nut_long  := 0.0;
nut_obliq := 0.0;

FOR i:=0 TO 62 DO
	nut_long  := nut_long  + 0.0001*( (sdelt[i]*t + sin_lng[i])*sarg[i]);
	nut_obliq := nut_obliq + 0.0001*( (cdelt[i]*t + cos_lng[i])*carg[i]);
END_FOR

END_FUNCTION_BLOCK

// ---- POUs/Functions/POLY.TcPOU
FUNCTION POLY : LREAL
VAR_INPUT
	// independent variable
	X:	LREAL;
END_VAR
VAR_IN_OUT
	// array of coefficients
	COEFFS: ARRAY [*] OF LREAL;
END_VAR
VAR
	i: DINT;
END_VAR

POLY := 0.0;
FOR i := LOWER_BOUND(COEFFS,1) TO UPPER_BOUND(COEFFS,1) DO
	POLY := POLY + COEFFS[i]*EXPT(X, i);
END_FOR

END_FUNCTION

// ---- POUs/FunctionBlocks/CO_ABERRATION.TcPOU
FUNCTION_BLOCK CO_ABERRATION
VAR_INPUT
	jd, 				// Julian Date
	ra, dec: LREAL; 	//ra and dec in degrees
	eps : LREAL := 0.0;
END_VAR
VAR_OUTPUT
	d_ra, d_dec: LREAL;
END_VAR
VAR
	sunpos: FB_SUNPOS;
	nutate: FB_NUTATE;
	sunra, sundec, sunlon,
	d_psi, d_epsilon, eps0,
	t, e, peri, cd, sd, ce, te, cp, sp, cs, ss, ca, sa, term1, term2, term3, term4: LREAL;
END_VAR
VAR CONSTANT
	d2r : LREAL := PI/180.0;
	k: LREAL := 20.49552; //constant of aberration, in arcseconds
	
END_VAR

(*
;+
;  NAME:
;     CO_ABERRATION
; PURPOSE:
;     Calculate changes to Ra and Dec due to the effect of annual aberration 
; EXPLANATION:
;      as described in Meeus, Chap 23.
; CALLING SEQUENCE:
;      co_aberration, jd, ra, dec, d_ra, d_dec, [EPS = ]
; INPUTS
;       jd      : Julian Date [scalar or vector]
;       ra, dec : Arrays (or scalars) of the ra  and dec's in degrees
;   Note: if jd is a vector, then ra and dec must either be scalars, or 
;                vectors of the same length.
;
; OUTPUTS
;       d_ra, d_dec: the corrections to ra and dec due to aberration in 
;                    arcseconds.  (These values can be added to the true RA 
;                    and dec to get the apparent position).   Note that d_ra
;                     is *not* multiplied by cos(dec), so that 
;                     apparent_ra = ra + d_ra/3600. 
; OPTIONAL INPUT KEYWORD:
;       eps : set this to the true obliquity of the ecliptic (in radians), or
;         it will be set for you if you don't know it (in that case, set it to
;                 an empty variable).
; EXAMPLE:
;   Compute the change in RA and Dec of Theta Persei (RA = 2h46m,11.331s, Dec =
;   49d20',54.54") due to aberration on 2028 Nov 13.19 TD
;
;      IDL> jdcnv,2028,11,13,.19*24,jd      ;Get Julian date
;      IDL> co_aberration,jd,ten(2,46,11.331)*15,ten(49,20,54.54),d_ra,d_dec
;
;      ==> d_ra = 30.045" (=2.003s)    d_dec = 6.697"
; NOTES:
;  These formula are from Meeus, Chapters 23.  Accuracy is much better than 1 
;   arcsecond.
;
;   The maximum deviation due to annual aberration is 20.49" and occurs when the
;   Earth velocity is perpendicular to the direction of the star.
;
; REVISION HISTORY:
;   Written, June 2002,      Chris O'Dell, U. of Wisconsin
;   Fix error with vector input   W. Landsman   June 2009
;   June 2009 update fixed case where JD was scalar but RA,Dec were vectors, but 
;     broke the case when both JD and RA,Dec were vectors Aug 2012 W. Landsman
;   Further fix when JD is 1 element vector  W. Landsman
;-
*)

T := (jd -2451545.0)/36525.0; // julian centuries from J2000 of jd.

IF EPS = 0.0 THEN
	// must calculate obliquity of ecliptic
	nutate(jd := jd, nut_long => d_psi, nut_obliq => d_epsilon); //d_psi and d_epsilon in degrees
	eps0 := ten(23,26,21.448)*3600.0 - 46.8150*T - 0.00059*EXPT(T, 2) +  0.001813*EXPT(T, 3);
	// TRUE obliquity OF the ecliptic in radians
	eps := (eps0 + d_epsilon)/3600.0*d2r; 	
END_IF

sunpos( JD := jd, RA => sunra, Dec => sundec, longmed => sunlon);

// Earth's orbital eccentricity
e := 0.016708634 - 0.000042037*T - 0.0000001267*EXPT(T, 2);
// longitude of perihelion, in degrees 
peri := 102.93735 + 1.71946*T + 0.00046*EXPT(T, 2);

//Useful Trig Functions
cd := COS(dec*d2r);		sd := SIN(dec*d2r);
ce := COS(eps); 		te := TAN(eps);
cp := COS(peri*d2r);	sp := SIN(peri*d2r);
cs := COS(sunlon*d2r);	ss := SIN(sunlon*d2r);
ca := COS(ra*d2r);		sa := SIN(ra*d2r);

term1 := (ca*cs*ce + sa*ss)/cd;
term2 := (ca*cp*ce + sa*sp)/cd;
term3 := (cs*ce*(te*cd - sa*sd) + ca*sd*ss);
term4 := (cp*ce*(te*cd - sa*sd) + ca*sd*sp);

d_ra := -k * term1 + e*k * term2;
d_dec := -k * term3 + e*k * term4;

END_FUNCTION_BLOCK

// ---- POUs/FunctionBlocks/FB_SUNPOS.TcPOU
FUNCTION_BLOCK FB_SUNPOS
VAR_INPUT
	// Julian Date
	JD:		LREAL;
	// output in Radians instead of Degrees
	RADIAN:	BOOL:= FALSE;
END_VAR
VAR_OUTPUT
	// right ascension
	RA,
	// declination of the sun
	Dec,
	// longitude
	longmed,
	// True Obliquity
	oblt:	LREAL;
END_VAR
VAR
	t, //  Julian centuries FROM 1900.0
	l, //  sun's mean longitude
	me, // Earth's mean anomaly
	ellcor, // ellipticity of the orbit
	mv, // mean anomaly of Venus
	vencorr,
	mm, 
	marscorr,
mj, jupcorr,
d, longterm, mooncorr,  omega:	LREAL;
END_VAR
VAR CONSTANT
	dtor: LREAL := PI/180.0; // Pi/180
END_VAR

(* source: https://idlastro.gsfc.nasa.gov/ftp/pro/astro/sunpos.pro *)

//  form TIME in Julian centuries FROM 1900.0
t := (jd - 2415020.0)/36525.0;

//  form sun's mean longitude
l := (279.696678+LMOD(36000.768925*t, 360.0))*3600.0;

//  allow for ellipticity of the orbit (equation of centre) using the Earth's mean anomaly ME
me := 358.475844 + LMOD(35999.049750*t, 360.0);
ellcor  := (6910.1 - 17.2*t)*SIN(me*dtor) + 72.3*SIN(2.0*me*dtor);
l := l + ellcor;
 
// allow FOR the Venus perturbations using the mean anomaly OF Venus MV
mv := 212.603219 + LMOD(58517.803875*t, 360.0);
vencorr := 4.8 * COS((299.1017 + mv - me)*dtor) + 
          5.5 * COS((148.3133 +  2.0 * mv  -  2.0 * me )*dtor) + 
          2.5 * COS((315.9433 +  2.0 * mv  -  3.0 * me )*dtor) + 
          1.6 * COS((345.2533 +  3.0 * mv  -  4.0 * me )*dtor) + 
          1.0 * COS((318.15   +  3.0 * mv  -  5.0 * me )*dtor);
l := l + vencorr;

//  Allow FOR the Mars perturbations using the mean anomaly OF Mars MM
mm := 319.529425  +  LMOD( 19139.858500 * t,  360.0 );
marscorr := 2.0 * COS((343.8883 -  2.0 * mm  +  2.0 * me)*dtor ) + 
            1.8 * COS((200.4017 -  2.0 * mm  + me) * dtor);
l := l + marscorr;

// Allow FOR the Jupiter perturbations using the mean anomaly OF Jupiter MJ
mj := 225.328328  +  LMOD( 3034.6920239 * t,  360.0 );
jupcorr := 7.2 * COS(( 179.5317 - mj + me )*dtor) + 
          2.6 * COS((263.2167  -  MJ ) *dtor) + 
          2.7 * COS(( 87.1450  -  2.0 * mj  +  2.0 * me ) *dtor) + 
          1.6 * COS((109.4933  -  2.0 * mj  +  me ) *dtor);
l := l + jupcorr;

// Allow FOR the Moons perturbations using the mean elongation OF the Moon from the Sun D
d := 350.7376814  + LMOD( 445267.11422 * t,  360.0 );
mooncorr  := 6.5 * SIN(d*dtor);
l := l + mooncorr;

// Allow for long period terms
longterm := 6.4 * SIN(( 231.19  +  20.20 * t )*dtor);
l :=  l + longterm;
l :=  LMOD( l + 2592000.0,  1296000.0); 
longmed := l/3600.0;

// Allow for Aberration
l :=  l - 20.5;

// Allow for Nutation using the longitude of the Moons mean node OMEGA
omega := 259.183275 - LMOD( 1934.142008 * t, 360.0);
l :=  l - 17.2 * SIN(omega*dtor);

// Form the True Obliquity
oblt := 23.452294 - 0.0130125*t + (9.2*COS(omega*dtor))/3600.0;

// Form Right Ascension AND Declination
l := l/3600.0;
//ra := ATAN2( COS(l*dtor), SIN(l*dtor) * COS(oblt*dtor));
ra := ATAN2( SIN(l*dtor) * COS(oblt*dtor), COS(l*dtor));
dec := ASIN(SIN(l*dtor) * SIN(oblt*dtor));
 
IF RADIAN THEN
	oblt := oblt*dtor; 
	longmed := longmed*dtor;
ELSE // result in degrees
	ra := MODABS(ra/dtor, 360.0);
    dec := dec/dtor;
END_IF

END_FUNCTION_BLOCK

// ---- POUs/Functions/TEN.TcPOU
FUNCTION TEN : LREAL
VAR_INPUT
	dd,mm,ss: LREAL;
END_VAR
VAR
END_VAR

TEN := dd + (mm/60.0) + (ss/3600.0);

END_FUNCTION

// ---- POUs/FunctionBlocks/CO_REFRACT.TcPOU
FUNCTION_BLOCK CO_REFRACT
VAR_INPUT
	old_alt: LREAL;
	altitude: LREAL := 0.0;
	pressure: LREAL := 0.0;
	temperature: LREAL := 0.0;
	epsilon: LREAL := 0.25; //accuracy of iteration for observed=TRUE case, in arcseconds
	TO_OBSERVED: BOOL;
END_VAR
VAR_OUTPUT
	new_alt: LREAL;
END_VAR
VAR
	aout, P, T, dr, cur, last : LREAL;
END_VAR
VAR CONSTANT
	alpha : LREAL := 0.0065; //temp lapse rate [deg C per meter]
END_VAR

IF temperature = 0.0 THEN
	IF altitude > 11000.0 THEN 
		temperature := 211.5; 
	ELSE 
		temperature := 283.0 - alpha*altitude;
	END_IF
END_IF

// estimate Pressure based on altitude, using U.S. Standard Atmosphere formula.
IF pressure = 0 THEN 
	pressure := 1010.0*EXPT(1-6.5/288000*altitude, 5.255);
END_IF

IF NOT TO_OBSERVED THEN 
	aout := old_alt - co_refract_forward(old_alt, P:=pressure,T:=temperature);
ELSE
	aout := 0.0;
	P := pressure; T := temperature;
	//calculate initial refraction guess
	dr := co_refract_forward(old_alt, P:=P, T:=T);
	cur := old_alt + dr; // guess of observed location

	REPEAT 
	 	last := cur;
		dr := co_refract_forward(cur, P:= P, T:=T);
	  	cur := old_alt + dr;
	UNTIL ABS(last-cur)*3600.0 < epsilon
	END_REPEAT
	aout := cur;
END_IF

new_alt := aout;

END_FUNCTION_BLOCK

// ---- POUs/Functions/CO_REFRACT_FORWARD.TcPOU
FUNCTION CO_REFRACT_FORWARD : LREAL
VAR_INPUT
	// The observed (apparent) altitude, in DEGREES.
	a: LREAL;
	// Pressure [in millibars]. Default is 1010 millibars.
	P: LREAL := 1010.0;
	// Ground Temp [in Celsius].  Default is 0 Celsius.
	T: LREAL := 0.0;
END_VAR
VAR
	Ref, tpcor: LREAL;
END_VAR
VAR CONSTANT
	d2r : LREAL := PI/180.0;
END_VAR

a := LIMIT(0.0, a, 90.0);
P := LIMIT(600.0, P, 1200.0);
T := LIMIT(-40.0, T, 40.0);

IF a >= 15.0 THEN
	Ref := 1.0 / TAN((a + 7.31/(a+4.4))*d2r);
ELSE
	Ref := 3.569*(0.1594 + 0.0196*a + 0.00002*EXPT(a, 2))/(1.0+0.505*a + 0.0845*EXPT(a, 2));
END_IF
tpcor := P * 283.15 / (1010.0 * (273.15 + T));
CO_REFRACT_FORWARD := tpcor * Ref;

END_FUNCTION

// ---- POUs/FunctionBlocks/FB_PRECESS.TcPOU
FUNCTION_BLOCK FB_PRECESS
VAR_INPUT
	ra, 
	dec,
	equinox1,
	equinox2: LREAL;
	RADIAN:	BOOL := FALSE;
END_VAR
VAR_OUTPUT
	ra_precessed,
	dec_precessed:	LREAL;
END_VAR
VAR
	ra_rad, dec_rad: LREAL;
	a,b,c,t: LREAL;
	x, x2: ARRAY[0..2] OF LREAL;
	st1: LREAL;
	rot: ARRAY[0..2,0..2] OF LREAL;
	sina, sinb, sinc, cosa,cosb,cosc: LREAL;
END_VAR
VAR CONSTANT
	deg_to_rad : LREAL := PI/180.0;
	sec_to_rad : LREAL := deg_to_rad/3600.0;
END_VAR

IF NOT RADIAN THEN
	ra_rad := ra*deg_to_rad;
	dec_rad := dec*deg_to_rad;
ELSE
    //Convert TO double precision IF NOT already
	ra_rad := ra;
	dec_rad := dec;
END_IF

a := COS( dec_rad );
x[0] := a*COS(ra_rad); x[1] := a*SIN(ra_rad); x[2] := SIN(dec_rad);

//*** PREMAT code starts here
ST1 := 0.001*( equinox1 - 2000.0);
t := 0.001*( equinox2 - equinox1);
//  Compute 3 rotation angles
A := sec_to_rad * T * (23062.181 + ST1*(139.656 +0.0139*ST1) + T*(30.188 - 0.344*ST1+17.998*T));
B := sec_to_rad * T * T * (79.280 + 0.410*ST1 + 0.205*T) + A;
C := sec_to_rad * T * (20043.109 - ST1*(85.33 + 0.217*ST1) + T*(-42.665 - 0.217*ST1 -41.833*T));
  sina := SIN(a); sinb := SIN(b);  sinc := SIN(c);
  cosa := COS(a); cosb := COS(b);  cosc := COS(c);

rot[0,0] :=  cosa*cosb*cosc-sina*sinb; 	rot[0,1] := sina*cosb+cosa*sinb*cosc; 	rot[0,2] := cosa*sinc;
rot[1,0] := -cosa*sinb-sina*cosb*cosc; 	rot[1,1] := cosa*cosb-sina*sinb*cosc; 	rot[1,2] := -sina*sinc;
rot[2,0] := -cosb*sinc;					rot[2,1] := -sinb*sinc; 				rot[2,2] := cosc;

//*** PREMAT code ends here

//x2 := rot* x; //rotate to get output direction cosines
x2[0] := rot[0,0]*x[0] + rot[1,0]*x[1] + rot[2,0]*x[2];
x2[1] := rot[0,1]*x[0] + rot[1,1]*x[1] + rot[2,1]*x[2];
x2[2] := rot[0,2]*x[0] + rot[1,2]*x[1] + rot[2,2]*x[2];

ra_rad := atan2(x2[1],x2[0]);
dec_rad := ASIN(x2[2]);

IF NOT RADIAN THEN
	ra_precessed := ra_rad/deg_to_rad;
	ra_precessed := MODABS(ra_precessed, 360.0);            //RA between 0 AND 360 degrees
	dec_precessed := dec_rad/deg_to_rad;
ELSE
	ra_precessed := ra_rad; 
	dec_precessed := dec_rad;
	ra_precessed := MODABS(ra_rad, 2.0*PI);
END_IF

END_FUNCTION_BLOCK

// ---- POUs/FunctionBlocks/FB_ALTAZ2HADEC.TcPOU
FUNCTION_BLOCK FB_ALTAZ2HADEC
VAR_INPUT
	// the local apparent altitude, in DEGREES
	alt:	LREAL;
	// the local apparent azimuth, in DEGREES
	az:		LREAL;
	// the local geodetic latitude, in DEGREES
	lat: 	LREAL;
END_VAR
VAR_OUTPUT
	// the local apparent hour angle, in DEGREES
	ha:		LREAL;
	// the local apparent declination, in DEGREES
	dec:	LREAL;
END_VAR
VAR
	alt_r:	LREAL;
	az_r:	LREAL;
	lat_r:	LREAL;
	sindec: LREAL;
END_VAR
VAR CONSTANT
	d2r:	LREAL := PI/180.0;
	//r2d:	LREAL := 180.0/PI;
	//h2r:	LREAL := PI/12.0;
	//h2d:	LREAL := 15.0;
END_VAR

(*

  NAME:
    ALTAZ2HADEC
 PURPOSE:
    Convert Horizon (Alt-Az) coordinates to Hour Angle and Declination.
 EXPLANATION::
    Can deal with the NCP singularity.    Intended mainly to be used by
    program hor2eq.pro
 CALLING SEQUENCE:
   ALTAZ2HADEC, alt, az, lat, ha, dec

 INPUTS
   alt - the local apparent altitude, in DEGREES, scalar or vector
   az  - the local apparent azimuth, in DEGREES, scalar or vector,
         measured EAST of NORTH!!!  If you have measured azimuth west-of-south
        (like the book MEEUS does), convert it to east of north via:
                       az = (az + 180) mod 360

   lat -  the local geodetic latitude, in DEGREES, scalar or vector.

 OUTPUTS
   ha  -  the local apparent hour angle, in DEGREES.  The hour angle is the 
          time that right ascension of 0 hours crosses the local meridian.  
          It is unambiguously defined.
   dec -  the local apparent declination, in DEGREES.

 EXAMPLE:
     Arcturus is observed at an apparent altitude of 59d,05m,10s and an 
     azimuth (measured east of north) of 133d,18m,29s while at the 
     latitude of +43.07833 degrees.
     What are the local hour angle and declination of this object?

     IDL> altaz2hadec, ten(59,05,10), ten(133,18,29), 43.07833, ha, dec
     ===> Hour angle ha = 336.683 degrees
          Declination, dec = 19.1824 degrees

       The widely available XEPHEM code gets:
                 Hour Angle = 336.683
                 Declination = 19.1824

 REVISION HISTORY:
    Written  Chris O'Dell Univ. of Wisconsin-Madison May 2002
*)
alt_r  := alt*d2r;
az_r := az*d2r;
lat_r := lat*d2r;

//******************************************************************************
// find local HOUR ANGLE (in degrees, from 0. to 360.)
ha := atan2( -SIN(az_r)*COS(alt_r), 
           -COS(az_r)*SIN(lat_r)*COS(alt_r)+SIN(alt_r)*COS(lat_r));
ha := ha / d2r;
IF ha < 0.0 THEN 
	ha := ha + 360.0;
END_IF
 ha := MODABS(ha, 360.0);

// Find declination (positive if north of Celestial Equator, negative if south)
sindec := SIN(lat_r)*SIN(alt_r) + COS(lat_r)*COS(alt_r)*COS(az_r);
// convert dec to degrees
dec := ASIN(sindec)/d2r;

END_FUNCTION_BLOCK

// ---- POUs/Functions/CT2LST.TcPOU
FUNCTION CT2LST : LREAL
VAR_INPUT
	lng: LREAL; // The longitude in degrees (east of Greenwich) of the place for which the local sidereal time is desired, scalar.   The Greenwich mean sidereal time (GMST) can be found by setting Lng = 0.
	jd:	LREAL; // this is the Julian date of time in question
END_VAR
VAR
	t0,t,theta: LREAL;
END_VAR
VAR CONSTANT
	jd2000: LREAL := 2451545.0;
END_VAR

(* source https://idlastro.gsfc.nasa.gov/ftp/pro/astro/ct2lst.pro 

;+
; NAME:
;     CT2LST
; PURPOSE:
;     To convert from Local Civil Time to Local Mean Sidereal Time.
;
; CALLING SEQUENCE:
;     CT2LST, Lst, Lng, Tz, Time, [Day, Mon, Year] 
;                       or
;     CT2LST, Lst, Lng, dummy, JD
;
; INPUTS:
;     Lng  - The longitude in degrees (east of Greenwich) of the place for 
;            which the local sidereal time is desired, scalar.   The Greenwich 
;            mean sidereal time (GMST) can be found by setting Lng = 0.
;     Tz  - The time zone of the site in hours, positive East  of the Greenwich
;           meridian (ahead of GMT).  Use this parameter to easily account 
;           for Daylight Savings time (e.g. -4=EDT, -5 = EST/CDT), scalar
;           This parameter is not needed (and ignored) if Julian date is 
;           supplied.    ***Note that the sign of TZ was changed in July 2008
;           to match the standard definition.*** 
;     Time or JD  - If more than four parameters are specified, then this is 
;               the time of day of the specified date in decimal hours.  If 
;               exactly four parameters are specified, then this is the 
;               Julian date of time in question, scalar or vector
;
; OPTIONAL INPUTS:
;      Day -  The day of the month (1-31),integer scalar or vector
;      Mon -  The month, in numerical format (1-12), integer scalar or vector
;      Year - The 4 digit year (e.g. 2008), integer scalar or vector
;
; OUTPUTS:
;       Lst   The Local Sidereal Time for the date/time specified in hours.
;
; RESTRICTIONS:
;       If specified, the date should be in numerical form.  The year should
;       appear as yyyy.
;
; PROCEDURE:
;       The Julian date of the day and time is question is used to determine
;       the number of days to have passed since 0 Jan 2000.  This is used
;       in conjunction with the GST of that date to extrapolate to the current
;       GST; this is then used to get the LST.    See Astronomical Algorithms
;       by Jean Meeus, p. 84 (Eq. 11-4) for the constants used.
;
; EXAMPLE:
;       Find the Greenwich mean sidereal time (GMST) on 2008 Jul 30 at 15:53 pm
;       in Baltimore, Maryland (longitude=-76.72 degrees).   The timezone is 
;       EDT or tz=-4
;
;       IDL> CT2LST, lst, -76.72, -4,ten(15,53), 30, 07, 2008
;
;               ==> lst =  11.356505  hours  (= 11h 21m 23.418s)
;
;       The Web site  http://tycho.usno.navy.mil/sidereal.html contains more
;       info on sidereal time, as well as an interactive calculator.
; PROCEDURES USED:
;       jdcnv - Convert from year, month, day, hour to julian date
;
; MODIFICATION HISTORY:
;     Adapted from the FORTRAN program GETSD by Michael R. Greason, STX, 
;               27 October 1988.
;     Use IAU 1984 constants Wayne Landsman, HSTX, April 1995, results 
;               differ by about 0.1 seconds  
;     Longitudes measured *east* of Greenwich   W. Landsman    December 1998
;     Time zone now measure positive East of Greenwich W. Landsman July 2008
;     Remove debugging print statement  W. Landsman April 2009
;-

*)

t0 := jd - jd2000;
t := t0/36525.0;
// Compute GST in seconds.
theta := 280.46061837 + (360.98564736629 * t0) + EXPT(t, 2)*(0.000387933 - (t/ 3871.0E4));
//theta := 100.46061837 + 36000.770053608*t0 + 0.000387933*EXPT(t0,2) - EXPT(t0,3)/3871000.0;
// Compute LST in hours.
CT2LST := ( theta + lng)/15.0;
CT2LST := MODABS(CT2LST, 24.0);

END_FUNCTION

// ---- POUs/TelescopeAuxiliary.TcPOU
PROGRAM TelescopeAuxiliary
VAR
	MQTTTimer : TON := (PT:=T#5S);
	pressure_voltage:	REAL;
END_VAR
VAR_OUTPUT
	// BT9 mirror
	temperature_mirror2:	REAL;
	// BT10
	temperature_mirror1:	REAL;
	// BT11

	// dewar pressure 0..10V Pfeiffer 
	pressure_Dewar:	REAL;
	// dewar temperature PT100
	temperature_Dewar:	REAL;
	

END_VAR

temperature_mirror2 := GVL_Telescope.temperature_mirror2 / 100.0;
temperature_mirror1 := GVL_Telescope.temperature_mirror1 / 100.0;

MQTTTimer(IN:=TRUE);
IF MQTTTimer.Q THEN // publish new payload every second

	MAIN.MQTTClient.Publish('telescope', 'dome',  'Mirror2Temperature',	LREAL_TO_FMTSTR(temperature_mirror2, 2, TRUE));
	MAIN.MQTTClient.Publish('telescope', 'dome', 'Mirror1Temperature',	LREAL_TO_FMTSTR(temperature_mirror1, 2, TRUE));
	
	MAIN.MQTTClient.Publish('telescope', 'instrument', 'DewarPressureVoltage',	LREAL_TO_FMTSTR(pressure_voltage, 3, TRUE));
	IF NOT GVL_Auxiliary.Dewar_temperature_error THEN
		MAIN.MQTTClient.Publish('telescope', 'instrument', 'DewarTemperature',	LREAL_TO_FMTSTR(temperature_Dewar, 2, TRUE));
	END_IF
	IF pressure_voltage > 0.001 THEN
		MAIN.MQTTClient.Publish('telescope', 'instrument', 'DewarPressure',	LREAL_TO_FMTSTR(pressure_Dewar, 2, TRUE));
	END_IF
	
	MQTTTimer(IN:=FALSE);

END_IF

END_PROGRAM

// ---- POUs/Functions/DateTime2JD.TcPOU
FUNCTION DateTime2JD : LREAL
VAR_INPUT
	epoch: TIMESTRUCT;
END_VAR
VAR
	a,y,m,d,jdn: LREAL;
END_VAR

(*    import datetime
    from math import floor
    if not type(epoch) is datetime.datetime:
        raise TypeError('datetime must be of type datetime')
    
    a = floor((14 - epoch.month)/12)
    y = epoch.year + 4800 - a
    m = epoch.month + 12*a - 3
    
    d = epoch.day
    d += epoch.hour/24. + epoch.minute/1440. + epoch.second/86400. # microsecond might be added here?
    
    if [epoch.year,epoch.month,d] >= [1582,10,15]:
        jdn = epoch.day + floor((153*m + 2)/5) + 365*y + floor(y/4) - floor(y/100) + floor(y/400) - 32045
    elif [epoch.year,epoch.month,d] <= [1582,10,4]:
        jdn = epoch.day + floor((153*m + 2)/5) + 365*y + floor(y/4) - 32083
    return jdn + (epoch.hour-12)/24. + epoch.minute/1440. + epoch.second/86400.
*)
a := FLOOR((14.0 - epoch.wMonth)/12.0);
y := epoch.wYear + 4800.0 - a;
m := epoch.wMonth + 12.0*a - 3.0;

d := epoch.wDay + (epoch.wHour/24.0) + (epoch.wMinute/1440.0) + (epoch.wSecond/86400.0);

//IF (epoch.wYear > 1582) (* AND (epoch.wMonth > 10.0) AND (d > 15.0)*) THEN
	jdn := epoch.wDay + FLOOR((153*m + 2)/5) + 365.0*y + FLOOR(y/4) - FLOOR(y/100) + FLOOR(y/400) - 32045.0;
//ELSIF (epoch.wYear < 1582) AND (epoch.wMonth < 10) AND (d > 4.0) THEN
//	jdn := epoch.wDay + FLOOR((153*m + 2)/5) + 365.0*y + FLOOR(y/4) - 32083.0;
//END_IF

DateTime2JD := jdn
			+ (epoch.wHour-12.0)/24.0
			+ (epoch.wMinute/1440.0) 
			+ (epoch.wSecond/86400.0)
			+ (DWORD_TO_REAL(epoch.wMilliseconds)/86400000.0);

END_FUNCTION

// ---- POUs/ElevationControl.TcPOU
PROGRAM ElevationControl
VAR_INPUT
	// increase the eleveation
	up:			BOOL;
	// decrease the elevation
	down:		BOOL;
	// reset an error
	reset:		BOOL;
	// enable the axis
	enable: 	BOOL;
	// set position of the axis in degrees
	position:	LREAL;
	// move axis command
	MoveAxis:	BOOL;
	// calibrate the focus axis
	HomeAxis:	BOOL;
	// enable tracking
	Tracking:	BOOL;
END_VAR
VAR_OUTPUT
	// axis is ready to operate
	Ready:			BOOL;
	// drive error condition
	error: 			BOOL;
	// warning condition
	warning:		BOOL;
	// actual position of the elevation axis
	act_position: 	LREAL;
	// error ID of the elevation axis
	ErrorID: 		UDINT;
	// axis is calibrated
	Calibrated:		BOOL;
	// time to reach target position
	slewtime:		LREAL;
END_VAR
VAR
	ElevationAxis:			FB_Axis2;
	ElevationCalibration: 	MC_SetPosition;
	fbSoEReset: 			FB_SoEReset;
	bSoEReset : BOOL;
	// delay until commutator angle is measured
	readydelay:				TON;
	getlastposition:		BOOL := TRUE;
	ElevationAxisEvent: 	FB_Eventlog;
	ElevationBrakeEvent: 	FB_Eventlog;
	HighElevationEvent: 	FB_Eventlog;
	LowElevationEvent:		FB_Eventlog;
	TorqueWarning:			FB_EventLog;
	CalibrationEvent:		FB_Eventlog;
	elevation_torque: REAL;
	ReadParameter:		MC_ReadParameter;
END_VAR
VAR CONSTANT
	// current position of the calibration cam. Apply an offset here if necessary
	calibration_position:	LREAL := 45.0;
END_VAR
VAR PERSISTENT
	last_position:	LREAL := -1.0;
END_VAR

// limit the position input to a sane value
position := LIMIT(0.0, position, 90.0);

//if we enable the axis, we have to open the brake first
IF Enable THEN
	HydraulicsControl.open_brake := TRUE;
END_IF

// if an error occurs on te enabled axis we close the brake
IF Enable AND error THEN
	Enable := FALSE;
	HydraulicsControl.close_brake := TRUE;
END_IF

IF ElevationAxis.Calibrated OR Error THEN
	HomeAxis := FALSE;
END_IF

Calibrated := ElevationAxis.Calibrated;

IF HomeAxis THEN
//	position := homing_position;
	position := calibration_position;
	MoveAxis := FALSE;
	Tracking := FALSE;
END_IF

IF MoveAxis THEN
	Tracking := FALSE;
END_IF

// if NOT Enabled and ActVelo>1 then issue a warning
warning := NOT enable AND GVL_Telescope.ElevationAxisRef.NcToPlc.ActVelo>2.0;

// deactivate limit switches on homing
MC_SetAcceptBlockedDriveSignal(
	Axis := GVL_Telescope.ElevationAxisRef, 
	Enable := HomeAxis);

IF Tracking AND ABS(position - act_position) > 1.0 THEN
	MoveAxis := TRUE;
END_IF

	
ElevationAxis(
	Enable := 			enable AND HydraulicsControl.brake_open,
	Reset := 			reset,
	MoveAxis :=			MoveAxis,
	HomeAxis :=			HomeAxis,
	Tracking :=			Tracking,
	Position := 		position, 
	Enable_Positive :=  GVL_Telescope.Elevation_inputs.0 OR HomeAxis,
	Enable_Negative := 	GVL_Telescope.Elevation_inputs.1,
	Jog_Forward :=		up,
	Jog_Backwards := 	down,
	bCalibrationCam :=	NOT GVL_Telescope.Elevation_inputs.0,
	ActualPosition => 	act_position,
	Error => 			error,
	ErrorID => 			ErrorID,
	AxisRef :=			GVL_Telescope.ElevationAxisRef);

IF ElevationAxis.MoveDone THEN
	MoveAxis := FALSE;
END_IF

IF ElevationAxis.HomeDone THEN
	HomeAxis := FALSE;
END_IF
	
IF ElevationAxis.ResetDone THEN
	reset := FALSE;
END_IF

ElevationCalibration(Axis := GVL_Telescope.ElevationAxisRef,
	Execute := getlastposition AND last_position>=0.0 AND NOT Calibrated,
	Position := last_position);

IF ElevationCalibration.Done THEN
	getlastposition := FALSE;
END_IF

IF Calibrated THEN
	last_position := act_position;
END_IF
	
bSoEReset := GVL_Telescope.Elevation_diagnostic = 16#0000F10B OR GVL_Telescope.Elevation_diagnostic = 16#0000F601;

IF bSoEReset THEN
	last_position := -1.0;
	fbSoEReset(
		Axis := GVL_Telescope.ElevationAxisRef,
		Execute := TRUE,
		Timeout := DEFAULT_ADS_TIMEOUT);
 	IF NOT fbSoEReset.Busy THEN
		fbSoEReset(Axis := GVL_Telescope.ElevationAxisRef, Execute := FALSE);
		bSoEReset := FALSE;
		Reset := TRUE;
	END_IF
END_IF 

readydelay(IN :=  HydraulicsControl.brake_open, PT := T#6000MS, Q=> ready);

ReadParameter(	Axis := GVL_Telescope.ElevationAxisRef, 
				Enable := ElevationAxis.InMotion, 
				ParameterNumber := MC_AxisParameter.AxisRemainingTimeToGo, 
				ReadMode := E_ReadMode.READMODE_CYCLIC);
				
IF ReadParameter.Valid THEN
	slewtime := ReadParameter.Value;
END_IF

elevation_torque := GVL_Telescope.Elevation_torque / 10.0;

		
ElevationAxisEvent(	Trigger := Error, 
				Level := ADSLOG_MSGTYPE_ERROR,
				FormatString := 'Elevation Axis Error: %s',
				OnMessage := NCError_TO_STRING(ErrorID));

HighElevationEvent(	Trigger := Calibrated AND act_position > 80.0, 
				Level := ADSLOG_MSGTYPE_WARN,
				FormatString := 'High Elevation: %s',
				OnMessage := LREAL_TO_FMTSTR(act_position, 2, TRUE));

LowElevationEvent(	Trigger := Calibrated AND act_position < 15.0, 
				Level := ADSLOG_MSGTYPE_WARN,
				FormatString := 'Low Elevation: %s',
				OnMessage := LREAL_TO_FMTSTR(act_position, 2, TRUE));
				
ElevationBrakeEvent( Trigger := NOT enable AND HydraulicsControl.brake_open, 
				Level := ADSLOG_MSGTYPE_WARN,
				FormatString := '%s',
				OnMessage := 'Brake was opened without elevation axis enabled!'); 

TorqueWarning(	
	Trigger := 		ABS(elevation_torque) > 60.0, 
	Level := 		ADSLOG_MSGTYPE_WARN,
	FormatString :=	'%s',
	OnMessage := 	'Elevation torque is high.');
	
CalibrationEvent(
	Trigger :=	Calibrated,
	Level :=	ADSLOG_MSGTYPE_HINT,
	OnMessage := 'Elevation is calibrated.'
	);

END_PROGRAM

// ---- POUs/FunctionBlocks/FB_Axis2.TcPOU
FUNCTION_BLOCK FB_Axis2
VAR_INPUT
	// enable the axis
	Enable:		BOOL;
	// reset the axis after error
	Reset: 		BOOL;
	// Move the Axis to a given position
	MoveAxis: 	BOOL;
	// HomeAxis;
	HomeAxis:	BOOL;
	// Stop the axis
	StopAxis:	BOOL;
	// position to move to
	Position: 	LREAL;
	// maximum velocity
	Velocity:	LREAL := 10.0;
	// Enable movement in positive direction (considering limit switch)
	Enable_Positive:	BOOL := TRUE;
	// Enable movement in negative direction (considering limit switch)
	Enable_Negative:	BOOL := TRUE;
	// jog forward
	Jog_Forward:		BOOL := FALSE;
	// jog backward
	Jog_Backwards:		BOOL := FALSE;
	// calibration input for homing
	bCalibrationCam:	BOOL;
	isModuloAxis:		BOOL := FALSE;
	// enable external setpoint generator
	Tracking:			BOOL;
	HomingMode:			MC_HomingMode := MC_HomingMode.MC_DefaultHoming;
END_VAR
VAR_OUTPUT
	// Reset has been executed
	ResetDone:	BOOL; 
	// the axis is in target position
	MoveDone:	BOOL;
	// the axis hass jogged
	JogDone:	BOOL;
	// the axis has stopped
	StopDone: 	BOOL;
	// the axis was calibrated and has come to a standstill
	HomeDone:	BOOL;
	// the axis is ready
	Ready:		BOOL;
	// the command has been aborted
	CommandAborted: BOOL;
	// axis busy
	Busy: 		BOOL;
	// axis is moving
	Active: 	BOOL;
	// axis is stopping
	Stopping:	BOOL;
	// axis is standing still (no commands issued) this should be the default
	StandStill:	BOOL;
	// axis is in motion
	InMotion:	BOOL;
	// axis is homing
	Homing:		BOOL;
	// axis is Accelerating or Decelerating
	InRamp:		BOOL;
	// axis is tracking on position
	isTracking:	BOOL;
	//	error condition
	Error: 		BOOL;
	// number of error
	ErrorID: 	UDINT;
	// actual position of the axis
	ActualPosition: LREAL;
	// axis is calibrated;
	Calibrated:	BOOL := FALSE;
	
END_VAR
VAR
	Axis_Power:		MC_Power;
	Axis_Reset:		MC_Reset;
	Axis_Move:		MC_MoveAbsolute;
	Axis_Modulo:	MC_MoveModulo;
	//Axis_Position:	MC_ReadActualPosition;
	Axis_Stop:		MC_Stop;
	Axis_Status:	MC_ReadStatus;
	Axis_Home:		MC_Home;
	Axis_Jog: 		MC_Jog;
	Axis_SetpointEnable:	MC_ExtSetPointGenEnable;
	Axis_SetpointDisable:	MC_ExtSetPointGenDisable;
	StopAllowed:	BOOL;
	// Direction for Axis_SetpointFeed
	Direction:			DINT;
	// difference between set position and measured position
	PositionDifference:	LREAL;
	TrackPosition:		LREAL;
	TrackVelocity:		LREAL;
	TrackAcceleration:	LREAL;
END_VAR

VAR_IN_OUT
	// axis reference
	AxisRef:	AXIS_REF;
END_VAR

// query the status of the axis at the beginning of the cycle
Axis_Status(Enable := TRUE,
			Axis := AxisRef);

// Enable the axis (power signal or manual enable)
Axis_Power(
	Axis := AxisRef,
	Enable := Enable,
	Enable_Positive := Enable_Positive,
	Enable_Negative := Enable_Negative,
	Override := 100.0,
	Status => Ready);

Axis_Reset(
	Axis := 	AxisRef,
	Execute := 	Reset,
	Done => 	ResetDone);

(* Tracking section ********************************************** *)

IF Tracking THEN
	PositionDifference := LIMIT(-0.002, Position - ActualPosition, 0.002);
	TrackPosition := ActualPosition + PositionDifference;
	TrackVelocity := 0.0; // LIMIT(-1.0, 2.0 * Velocity, 1.0);
	TrackAcceleration := 0.0;
ELSE
	TrackPosition := ActualPosition;
	TrackVelocity := 0.0;
	TrackAcceleration := 0.0;
END_IF


IF NOT Tracking OR ABS(PositionDifference) < 1E-5 THEN // TrackVelocity = 0 AND TrackAcceleration = 0 THEN
	Direction := 0;
ELSIF PositionDifference < 0.0 THEN
	Direction := -1;
ELSE
	Direction := 1;
END_IF

isTracking := Tracking AND ABS(Position - ActualPosition) < 5.0E-3;
IF Tracking AND Ready AND Calibrated AND NOT StopAxis THEN
	Axis_SetpointEnable.Execute := TRUE;
ELSIF NOT Axis_SetpointEnable.Busy AND Axis_SetpointEnable.Done THEN
	Axis_SetpointEnable.Execute := FALSE;
END_IF

Axis_SetpointEnable(Axis := AxisRef,
	Position :=		TrackPosition,	// final destination
	PositionType := POSITIONTYPE_ABSOLUTE);
	
MC_ExtSetPointGenFeed(
	Position :=		TrackPosition,
	Velocity :=		TrackVelocity,
	Acceleration :=	TrackAcceleration,
	Direction :=	Direction, 
	Axis :=			AxisRef);

Axis_SetpointDisable(Axis := AxisRef,
	Execute := NOT Tracking);
	
(* end of tracking section  ********************************************** *)
	
IF isModuloAxis THEN
	Axis_Modulo( 
		Axis := 		AxisRef,
		Execute := 		MoveAxis AND Ready AND Calibrated,
		Position := 	Position,
		Velocity :=		Velocity,
		Direction := 	MC_Shortest_Way,
		Done => 		MoveDone);
ELSE
	Axis_Move( 
		Axis := 		AxisRef,
		Execute := 		MoveAxis AND Ready AND Calibrated,
		Position := 	Position,
		Velocity := 	Velocity,
		Done => 		MoveDone);
END_IF

Axis_Jog(
	JogForward := 	Jog_Forward AND Ready AND Enable_Positive,
	JogBackwards := Jog_Backwards AND Ready AND Enable_Negative,
	Mode := 		MC_JOGMODE_STANDARD_FAST,
	Done => 		JogDone, 
	Axis := 		AxisRef);

Axis_Home(
	Axis := 			AxisRef,
	Execute := 			HomeAxis AND Ready,
	Position := 		position, //DEFAULT_HOME_POSITION,
	HomingMode :=		HomingMode,
	bCalibrationCam := 	bCalibrationCam,
	Done => 			HomeDone);	
(*	
IF (MoveDone OR HomeDone OR JogDone) AND NOT Axis_Status.StandStill THEN
	StopAxis := TRUE;
END_IF
*)
IF MoveDone AND (NOT Axis_Modulo.Busy OR NOT Axis_Move.Busy) THEN
	MoveAxis := FALSE;
END_IF

IF JogDone THEN
	Jog_Forward := FALSE;
	Jog_Backwards := FALSE;
END_IF

IF HomeDone THEN
	Calibrated := TRUE;
	HomeAxis := FALSE;
END_IF

IF StopDone THEN
	StopAxis := FALSE;
END_IF

StopAllowed :=	Axis_Status.StandStill OR  
				Axis_Status.ContinuousMotion OR
				Axis_Status.DiscreteMotion OR
				Axis_Status.SynchronizedMotion OR
				Axis_Status.Homing;

Axis_Stop( 
	Axis := 	AxisRef,
	Execute := 	StopAxis AND StopAllowed,
	Done => 	StopDone);
(*
Axis_Position(
	Axis := 	AxisRef,
	Enable := 	Calibrated,
	Position => AbsolutePosition);
*)
IF isModuloAxis THEN
	ActualPosition := AxisRef.NcToPlc.ModuloActPos; // required e.g. for Filterwheel
ELSE
	ActualPosition := AxisRef.NcToPlc.ActPos;
END_IF

IF Axis_Power.Error THEN
	ErrorID := Axis_Power.ErrorID;
END_IF

IF Axis_SetpointEnable.Error THEN
	ErrorID := Axis_SetpointEnable.ErrorID;
END_IF

IF Axis_Reset.Error THEN
	ErrorID := Axis_Reset.ErrorID;
END_IF

IF Axis_Modulo.Error THEN
	ErrorID := Axis_Modulo.ErrorID;
END_IF

IF Axis_Move.Error THEN
	ErrorID := Axis_Move.ErrorID;
END_IF

IF Axis_Home.Error THEN
	ErrorID := Axis_Home.ErrorID;
END_IF

IF Axis_Jog.Error THEN
	ErrorID := Axis_Jog.ErrorID;
END_IF

IF Axis_Stop.Error THEN
	ErrorID := Axis_Stop.ErrorID;
END_IF

Busy := 	Axis_SetpointEnable.Busy OR
			Axis_Reset.Busy OR 
			Axis_Modulo.Busy OR
			Axis_Move.Busy OR 
			Axis_Home.Busy OR
			Axis_Jog.Busy;

Error := 	Axis_Power.Error OR 
			Axis_SetpointEnable.Error OR
			Axis_Reset.Error OR 
			Axis_Modulo.Error OR
			Axis_Move.Error OR 
			Axis_Home.Error OR
			Axis_Jog.Error OR 
			Axis_Stop.Error;

Active := 	// Axis_Power.Active OR //alsways true if enabled 
			Axis_Modulo.Active OR
			Axis_Move.Active OR 
			Axis_Home.Active OR
			Axis_Jog.Active OR 
			Axis_Stop.Active;

CommandAborted :=	Axis_Modulo.CommandAborted OR
					Axis_Move.CommandAborted OR 
					Axis_Home.CommandAborted OR
					Axis_Jog.CommandAborted OR 
					Axis_Stop.CommandAborted;	
	
IF NOT Error THEN
	ErrorID := 0;
END_IF
			
InMotion := Axis_Status.ConstantVelocity OR
			Axis_Status.DiscreteMotion OR
			Axis_Status.ContinuousMotion OR
			Axis_Status.SynchronizedMotion; 
InRamp :=	Axis_Status.Accelerating OR
			Axis_Status.Decelerating;
Stopping := Axis_Status.Stopping;
StandStill := Axis_Status.StandStill;
Homing :=	Axis_Status.Homing;
// InPosition := AxisRef.NcToPlc.TargetPos;

END_FUNCTION_BLOCK

// ---- POUs/HydraulicsControl.TcPOU
PROGRAM HydraulicsControl
VAR_INPUT
	// start the hydraulics
	start:		BOOL := FALSE;
	// stop the hydraulics
	stop: 		BOOL;
	// command to open the brake
	open_brake:	BOOL := FALSE;
	// command to open the brake
	close_brake: BOOL;
	// reset any hydraulics error
	reset: 		BOOL;
END_VAR
VAR_OUTPUT
	// status of the brake: is the brake open?
	brake_open:			BOOL;
	// is the brake closed?
	brake_closed:		BOOL;
	// pump is running, but the pressure remains low
	pressure_failure:	BOOL;
	// suction was started, but it is not running
	suction_failure:	BOOL;
	// main pump is running but suction has a timeout
	hydraulics_failure:	BOOL;
	// oil is low
	oil_low:			BOOL;
	// oil is high (unused?)
	oil_high:			BOOL;
	// oil pressure is 25 bars
	oil_pressure_OK:	BOOL;
	// oil is on reserve
	oil_warning:		BOOL;
	// oil filter is dirty
	oil_filter_dirty:	BOOL;
	// oil is below 10°C
	oil_cold:			BOOL;
	// oil is above 50°C
	oil_hot:			BOOL;
	// main pump is running
	pump_running:		BOOL;
	// suction pump is running
	suction_running :	BOOL := FALSE;
	// error condition
	error: 				BOOL;
END_VAR
VAR
	// monitors the pressure of the pump is running
	pressure_watchdog:	TON;
	// monitors the activation of the suction pump
	suction_watchdog: TON;
	// watch the hydraulics and suction pumps
	hydraulics_watchdog: TON;
	// the suction pump is activated for at least 28s when maximum is reached
	suction_pump_timer: TP;
	// represents the state of the main pump
	oil_pump_state:		RS;
	// represents the state of the brake
	brake_state: 		RS;
	// wait for the brake to open after pressure has been established
	brake_open_delay:	TON;
	// report brake opend after a short delay
	brake_opened_delay:	TON;
	// error state (set dominant)
	error_state:	SR;
	HydraulicsLog,
	PumpLog,
	ReserveLog,
	oil_low_log,
	FilterLog,
	OverTemperatureLog,
	UnderTemperatureLog,
	SuctionLog,
	BreakClearingWarning,
	BreakHydraulicsWarning: FB_EventLog;
	
	// measures the operating cycle of the suction pump
	suction_timer : FB_Timer;
	pressure_timer:	TIMER;
	oil_pan_timer: TIMER;
	StatusWord, LastStatus:	UDINT;
END_VAR

(* 
Main control Logic for the Hydraulics system
* power on delay for main pump and suction pump
* start main pump if main control is ready (button pressed or remote)
* start suction pump if maximum in pan is reached
* suction pump runs for 60 seconds
* stop main pump if oil is low
* stop main pump if pressure fails for 10 seconds
*)
oil_low := NOT GVL_Hydraulics.oil_low;
oil_high := NOT GVL_Hydraulics.oil_high;
oil_warning := GVL_Hydraulics.oil_reserve;
oil_pressure_OK := GVL_Hydraulics.oil_pressure_OK;
oil_filter_dirty := NOT GVL_Hydraulics.oilfilter_dirty;
oil_cold := NOT GVL_Hydraulics.oil_undertemperature;
oil_hot := GVL_Hydraulics.oil_overtemperature;
pump_running := GVL_Hydraulics.pump_running;
suction_running := GVL_Hydraulics.suction_running;

IF stop THEN
	start := FALSE;
END_IF

error_state(SET1 := pressure_failure OR	suction_failure OR hydraulics_failure OR oil_low,
			RESET := reset,
			Q1 => error);

oil_pump_state(SET := start,
				RESET1 := stop OR error OR NOT MAIN.phase_available);

GVL_Hydraulics.oil_pump_enable := oil_pump_state.Q1;

IF NOT pump_running THEN
	stop := FALSE;
END_IF
(* This section controls the hydraulic brake responsible for azimuth and elevation. 
Especially the elevation is imbalanced if not in the position control loop. 
The brake must only be opened, if the elevation drive is activated concurrently.
*)
// reset the open_brake command if the close_brake is active


// wait for pressure to build up (hack for oil_pressure_ok)
brake_open_delay(IN := pump_running AND oil_pressure_OK,
				PT := T#3S);
//manually or remotly open brake. Close brake on limit switch. Wait n seconds after pump is on
//hold the brake, if we reach the az-limit	
// close the brake if the pump is not running	

IF close_brake OR NOT pump_running THEN 
	open_brake := FALSE;
END_IF
		
brake_state(SET := brake_open_delay.Q AND open_brake AND MAIN.brake_clearing,
			RESET1 := GVL_Telescope.azimut_limit_switch 
					  OR close_brake 
					  OR NOT pump_running
					  OR NOT MAIN.brake_clearing,
			Q1 => GVL_Telescope.brake_azimuth_eve);

brake_opened_delay(	IN :=brake_state.Q1, 
					PT := T#1000MS,
					Q => brake_open);

brake_closed := NOT brake_open;
IF brake_closed THEN
	close_brake := FALSE;
END_IF

(* This is the end of the brake control section *)

// measure suction pump cycle
suction_timer(	bStart := suction_running AND NOT suction_pump_timer.Q, 
				bStop := GVL_Hydraulics.oilpan_maximum);  

suction_pump_timer(IN := MAIN.phase_available AND 
						GVL_Hydraulics.oilpan_maximum,
					PT := T#48S,
					Q => GVL_Hydraulics.oil_suction_enable);
					
(*					
IF MAIN.phase_available AND GVL_Hydraulics.oilpan_maximum THEN 
  GVL_Hydraulics.oil_suction_enable := TRUE;
END_IF
					
IF MAIN.phase_available AND NOT suction_min_duration AND oil_warning THEN
  GVL_Hydraulics.oil_suction_enable := FALSE;
END_IF
*)	
					
suction_watchdog(IN := GVL_Hydraulics.oil_suction_enable AND NOT suction_running,
					PT := T#10S,
					Q => suction_failure);
					
pressure_watchdog(IN := GVL_Hydraulics.oil_pump_enable AND 
						NOT oil_pressure_OK,
					PT := T#15S,
				  Q => pressure_failure);
hydraulics_watchdog(IN := pump_running AND NOT suction_running,
						PT := T#140S,
						Q => hydraulics_failure);

pressure_timer(bStart := GVL_Hydraulics.oil_pump_enable AND NOT oil_pressure_OK);
oil_pan_timer(bStart := GVL_Hydraulics.oilpan_maximum AND suction_running);
						
StatusWord.0 := oil_low;
StatusWord.1 := oil_high;
StatusWord.2 := oil_warning;
StatusWord.3 := oil_pressure_OK;
StatusWord.4 := oil_filter_dirty;
StatusWord.5 := oil_cold;
StatusWord.6 := oil_hot;
StatusWord.7 := brake_open;
StatusWord.8 := GVL_Main.brake_clearing;
StatusWord.9 := pump_running;
StatusWord.10 := suction_running;
StatusWord.11 := GVL_Hydraulics.oilpan_maximum;


IF StatusWord<>LastStatus THEN // publish new payload every second
	LastStatus := StatusWord;
	MAIN.MQTTClient.Publish('hydraulics', 'base', 'OilLow',			BOOL_TO_STRING(oil_low));
	MAIN.MQTTClient.Publish('hydraulics', 'base', 'OilHigh',		BOOL_TO_STRING(oil_high));
	MAIN.MQTTClient.Publish('hydraulics', 'base', 'OilReserve',		BOOL_TO_STRING(oil_warning));
	MAIN.MQTTClient.Publish('hydraulics', 'base', 'OilPressureOK', 	BOOL_TO_STRING(oil_pressure_OK));
	MAIN.MQTTClient.Publish('hydraulics', 'base', 'OilFilterDirty',	BOOL_TO_STRING(oil_filter_dirty));
	MAIN.MQTTClient.Publish('hydraulics', 'base', 'OilCold',		BOOL_TO_STRING(oil_cold));
	MAIN.MQTTClient.Publish('hydraulics', 'base', 'OilHot',			BOOL_TO_STRING(oil_Hot));
	MAIN.MQTTClient.Publish('hydraulics', 'base', 'BrakeOpen',		BOOL_TO_STRING(brake_open));
	MAIN.MQTTClient.Publish('hydraulics', 'base', 'BrakeClearing',	BOOL_TO_STRING(GVL_Main.brake_clearing));
	MAIN.MQTTClient.Publish('hydraulics', 'base', 'PumpRunning',	BOOL_TO_STRING(pump_running));
	MAIN.MQTTClient.Publish('hydraulics', 'base', 'SuctionRunning',	BOOL_TO_STRING(suction_running));
	MAIN.MQTTClient.Publish('hydraulics', 'base', 'OilPanMaxiumum',	BOOL_TO_STRING(GVL_Hydraulics.oilpan_maximum));
	IF pressure_timer.valid THEN
		MAIN.MQTTClient.Publish('hydraulics', 'base', 'OilViscosity1',	INT_TO_STRING(TIME_TO_INT(pressure_timer.tDifference)));
	END_IF
	IF oil_pan_timer.valid THEN
		MAIN.MQTTClient.Publish('hydraulics', 'base', 'OilViscosity2',	INT_TO_STRING(TIME_TO_INT(oil_pan_timer.tDifference)));
	END_IF
END_IF


				  				  
HydraulicsLog(Trigger := pressure_failure,
				Level := ADSLOG_MSGTYPE_ERROR,
				FormatString := 'oil pressure: %s',
				OnMessage := 'FAILURE',
				OffMessage := 'OK',
				OffLevel := ADSLOG_MSGTYPE_HINT);

PumpLog(Trigger := pump_running,
				Level := ADSLOG_MSGTYPE_HINT,
				FormatString := 'Main hydraulics pump: %s',
				OnMessage := 'START',
				OffMessage := 'STOP',
				OffLevel := ADSLOG_MSGTYPE_HINT);
	
ReserveLog(Trigger := oil_warning,
			Level := ADSLOG_MSGTYPE_WARN,
			FormatString := 'oil reserve: %s',
			OnMessage := 'LOW',
			OffMessage := 'OK',
			OffLevel := ADSLOG_MSGTYPE_HINT);

oil_low_log(Trigger := oil_low,
				Level := ADSLOG_MSGTYPE_ERROR,
				FormatString := 'oil level: %s',
				OnMessage := 'LOW',
				OffMessage := 'OK',
				OffLevel := ADSLOG_MSGTYPE_HINT);

FilterLog(Trigger := oil_filter_dirty,
				Level := ADSLOG_MSGTYPE_WARN,
				FormatString := 'Hydraulics Filter is %s',
				OnMessage := 'dirty.');

OverTemperatureLog(Trigger := oil_hot,
				Level := ADSLOG_MSGTYPE_WARN,
				FormatString := 'Hydraulics Temperature is %s',
				OnMessage := 'high.');
UnderTemperatureLog(Trigger := oil_cold,
				Level := ADSLOG_MSGTYPE_WARN,
				FormatString := 'Hydraulics Temperature is %s',
				OnMessage := 'low.');

SuctionLog(Trigger := suction_failure OR hydraulics_failure,
				Level := ADSLOG_MSGTYPE_ERROR,
				FormatString := 'suction pump: %s',
				OnMessage := 'FAILURE',
				OffMessage := 'OK',
				OffLevel := ADSLOG_MSGTYPE_HINT);

BreakClearingWarning(Trigger := NOT Main.brake_clearing AND open_brake,
				Level := ADSLOG_MSGTYPE_WARN,
				FormatString := '%s',
				OnMessage := 'Cannot open brake without brake clearing.');

BreakHydraulicsWarning(Trigger := NOT start AND open_brake,
				Level := ADSLOG_MSGTYPE_WARN,
				FormatString := '%s',
				OnMessage := 'Cannot open brake without running hydraulics.');

END_PROGRAM

// ---- POUs/FunctionBlocks/FB_Timer.TcPOU
FUNCTION_BLOCK FB_Timer
VAR_INPUT
	bStart          : BOOL := FALSE;
	bStop			: BOOL := FALSE;
END_VAR
VAR_OUTPUT
    tDifference     : TIME;
END_VAR
VAR
    StartTrigger,
	StopTrigger		: R_TRIG;
    StartTime    	: TIME;
    StopTime    	: TIME;
END_VAR

(*
Timer functionblock

Source:
https://infosys.beckhoff.de/index.php?content=../content/1031/tc3_plc_intro/2529365899.html&id=
*)
StartTrigger(CLK := bStart);
StopTrigger(CLK := bStop);

IF StartTrigger.Q THEN
    StartTime  := TIME();
END_IF

IF StopTrigger.Q THEN
    StopTime  := TIME();
    tDifference   := StopTime - StartTime;    // The difference will be T#5s
END_IF

END_FUNCTION_BLOCK

// ---- POUs/FunctionBlocks/TIMER.TcPOU
FUNCTION_BLOCK TIMER
VAR_INPUT
	bStart:	BOOL := TRUE;
END_VAR
VAR_OUTPUT
	tDifference:	TIME;
	valid: 			BOOL;
END_VAR
VAR
	tTimeReturn1:	TIME;
	tTimeReturn2:	TIME;
	fbTrigger1:		R_TRIG;
	fbTrigger2:		F_TRIG;
END_VAR

fbTrigger1(CLK := bStart);
fbTrigger2(CLK := bStart);

IF fbTrigger1.Q THEN
	tTimeReturn1 := TIME();
	valid := FALSE;
END_IF

IF bStart OR fbTrigger2.Q THEN
	tTimeReturn2 := TIME();
END_IF

IF fbTrigger2.Q THEN
	valid := TRUE;
END_IF

tDifference := tTimeReturn2 - tTimeReturn1;

END_FUNCTION_BLOCK

// ---- POUs/Functions/NCError_TO_STRING.TcPOU
FUNCTION NCError_TO_STRING : STRING(255)
VAR_INPUT
	// NC Error ID
	ErrorID:	UDINT;
END_VAR
VAR
END_VAR

NCError_TO_STRING := '';

CASE ErrorID OF
	16#4220:	NCError_TO_STRING := 'Group not ready / group not ready for new task';
	16#4253:	NCError_TO_STRING := 'Reference cam became free too soon';
	16#4260:	NCError_TO_STRING := 'Controller enable';
	16#42EF:	NCError_TO_STRING := 'Axis is locked for motion commands because a stop command is still active';
	16#4466:	NCError_TO_STRING := 'Invalid IO data FOR more than n subsequent NC cycles (encoder)';
	16#4550: 	NCError_TO_STRING := 'Following error monitoring (position)';
	16#4650:	NCError_TO_STRING := 'Drive hardware not ready to operate';
	16#4B07:	NCError_TO_STRING := 'Timeout axis function block';
	16#4B09:	NCError_TO_STRING := 'Axis is not ready';
	16#4B0A:	NCError_TO_STRING := 'Error during referencing';
ELSE
	NCError_TO_STRING := DWORD_TO_HEXSTR(ErrorID, 4, FALSE);
END_CASE

END_FUNCTION

// ---- POUs/AzimuthElevationControl.TcPOU
PROGRAM AzimuthElevationControl
VAR_INPUT
	// decrease azimuth
	left:		BOOL;
	// increase azimuth
	right: 		BOOL;
	// reset the axis
	Reset: 		BOOL;
	// enable the axis and its position control loop
	Enable:		BOOL;
	// Move azimuth to given position
	MoveAxis:	BOOL;
	// Home the axis
	HomeAxis:	BOOL;
	// enable tracking
	Tracking:	BOOL;
	// position to move the axis to
	position: 	LREAL;
END_VAR
VAR_OUTPUT
	// error state of the axis
	error: 			BOOL;
	// error ID of the axis
	ErrorID:		UDINT;
	// actual_position of the axis
	act_position:	LREAL;
	// is the axis calibrated
	calibrated:		BOOL;
	// drive is ready
	ready:			BOOL;
	// time to reach target position
	slewtime:		LREAL;
END_VAR
VAR
	AzimuthAxis:		FB_Axis2;
	AzimuthCalibration: MC_SetPosition;
	fbSoEReset:			FB_SoEReset;
	AzimuthAxisEvent: 	FB_EventLog;
	// delay until commutator angle is measured
	readydelay:			TON;
	HomeDelay:			FB_TONTP;
	TorqueError:		TON := (PT := T#3S);
	azimuth_torque: 	REAL;
	TorqueWarning:		FB_EventLog;
	CalibrationEvent:	FB_Eventlog;
	ReadParameter:		MC_ReadParameter;
	getlastposition:	BOOL := TRUE;
	bSoEReset:			BOOL;
	azimuth_rest_timer:	TON;
	azimuth_at_rest:	BOOL;
END_VAR
VAR CONSTANT
	// reference position for homing
	// homing_position:		LREAL := 439.0; // was 442 - -21.21 = 463.21; 463 + 24 = 439
	// current position of the calibration cam encoder zero index. Apply an offset here if necessary
	calibration_position:	LREAL := 156.1195; // 393.0; 
END_VAR
VAR PERSISTENT
	last_position:	LREAL := -1.0;
END_VAR

(* Azimuth Axis control section
Power must be on and brake must be open for the axis to operate
*)

// generate the ready signal after enabling the drive
readydelay(IN :=  AzimuthAxis.Enable, PT := T#3000MS, Q=> ready);

// limit the input position angle
position := LIMIT(0.0, position, 450.0);

// conduct the calibrated signal
calibrated := AzimuthAxis.Calibrated;

IF Calibrated OR Error THEN
	HomeAxis := FALSE;
	getlastposition := FALSE;
END_IF
	
IF HomeAxis THEN
	position := calibration_position;
END_IF

(*
// move to calibration_position after homing
HomeDelay(IN := Calibrated, PT1 := T#5S, PT2 := T#100MS);
*)
IF HomeDelay.Q THEN
	position := calibration_position;
	MoveAxis := TRUE;
END_IF

// perform a recalibration on the last known position
AzimuthCalibration(
	Axis := GVL_Telescope.AzimuthAxisRef,
	Execute := getlastposition AND last_position>=0.0 AND NOT Calibrated,
	Position := last_position);

IF AzimuthCalibration.Done THEN
	getlastposition := FALSE;
END_IF

IF Calibrated THEN
	last_position := act_position;
END_IF

// enable the azimuth if not moved by the power chain. Sorry for the hack
azimuth_rest_timer(IN := HydraulicsControl.brake_open AND 
				(ABS(GVL_Telescope.AzimuthAxisRef.NcToPlc.ActVelo) < 0.01), PT := T#2S);
IF azimuth_rest_timer.Q THEN
	azimuth_at_rest := TRUE;
ELSIF HydraulicsControl.brake_closed THEN
	azimuth_at_rest := FALSE;
END_IF
	
// deactivate limit switches on homing
MC_SetAcceptBlockedDriveSignal(
	Axis := GVL_Telescope.AzimuthAxisRef, 
	Enable := HomeAxis);

AzimuthAxis(	
	Enable := 			enable AND azimuth_at_rest,
	Reset := 			reset,
	MoveAxis :=			MoveAxis,
	HomeAxis := 		HomeAxis,
	Tracking :=			Tracking,
	Position := 		position, 
	Enable_Positive := 	NOT GVL_Telescope.azimut_limit_switch AND (GVL_Telescope.Azimuth_inputs.1 OR HomeAxis),
	Enable_Negative := 	NOT GVL_Telescope.azimut_limit_switch AND GVL_Telescope.Azimuth_inputs.0,
	Jog_Forward :=		right,
	Jog_Backwards := 	left,
	bCalibrationCam :=	NOT GVL_Telescope.Azimuth_inputs.1,
	ActualPosition => 	act_position,
	Error => 			error,
	ErrorID => 			ErrorID,
	AxisRef :=			GVL_Telescope.AzimuthAxisRef);

bSoEReset := GVL_Telescope.Azimuth_diagnostic = 16#0000F10B OR GVL_Telescope.Azimuth_diagnostic = 16#0000F601;

IF bSoEReset THEN
	last_position := -1.0;
	fbSoEReset(
		Axis := GVL_Telescope.AzimuthAxisRef,
		Execute := TRUE,
		Timeout := DEFAULT_ADS_TIMEOUT);
 	IF fbSoEReset.Busy THEN
		fbSoEReset(Axis := GVL_Telescope.AzimuthAxisRef, Execute := FALSE);
	ELSE
		bSoEReset := FALSE;
		Reset := TRUE;
	END_IF
END_IF 
	
IF AzimuthAxis.MoveDone THEN
	MoveAxis := FALSE;
END_IF

IF AzimuthAxis.HomeDone THEN
	HomeAxis := FALSE;
END_IF
	
IF AzimuthAxis.ResetDone THEN
	reset := FALSE;
END_IF

ReadParameter(	Axis := GVL_Telescope.AzimuthAxisRef, Enable := AzimuthAxis.InMotion, 
				ParameterNumber := MC_AxisParameter.AxisRemainingTimeToGo, 
				ReadMode := E_ReadMode.READMODE_CYCLIC);
IF ReadParameter.Valid THEN
	slewtime := ReadParameter.Value;
END_IF

azimuth_torque := GVL_Telescope.Azimuth_torque / 10.0;
TorqueError(IN := ABS(azimuth_torque) > 50.0);


AzimuthAxisEvent(	
	Trigger := 		Error, 
	Level := 		ADSLOG_MSGTYPE_ERROR,
	FormatString :=	'Azimuth Axis Error: %s',
	OnMessage := 	NCError_TO_STRING(ErrorID));
	
TorqueWarning(	
	Trigger := 		TorqueError.Q, 
	Level := 		ADSLOG_MSGTYPE_WARN,
	FormatString :=	'%s',
	OnMessage := 	'Azimuth torque is high.');
	
CalibrationEvent(
	Trigger := 		Calibrated, 
	Level := 		ADSLOG_MSGTYPE_HINT,
	FormatString :=	'%s',
	OnMessage := 	'Azimuth axis is calibrated.');

END_PROGRAM

// ---- POUs/FunctionBlocks/FB_TONTP.TcPOU
FUNCTION_BLOCK FB_TONTP
VAR_INPUT
	IN :	BOOL;
	 PT1:	TIME := T#1000MS;
	 PT2:	TIME := T#1000MS;
END_VAR
VAR_OUTPUT
	Q:	BOOL;
END_VAR
VAR
	ton:	TON;
	tp:		TP;
END_VAR

ton(IN := IN, PT := PT1);
tp(IN := ton.Q, PT := PT2, Q => Q);

END_FUNCTION_BLOCK

// ---- POUs/FilterWheelControl.TcPOU
PROGRAM FilterWheelControl
VAR_INPUT
	// enable the axis
	Enable:				BOOL;
	// reset the axis(-error)
	Reset:				BOOL;
	// move counter-clockwise
	left:				BOOL;
	// move clockwise
	right:				BOOL;
	// TRUE, if the filter is in position and wheel has come to rest
	Ready:				BOOL;
	// filter position
	filter_position: 	WORD;
	// move to given position
	MoveAxis: 			BOOL;
	// calibrate the axis
	HomeAxis:			BOOL;
END_VAR
VAR_OUTPUT
	// is true if an error occurred
	error: 				BOOL;
	// number of current axis error
	ErrorID:			UDINT;
	act_position:		LREAL;
	// axis has been calibrated
	Calibrated :		BOOL;
END_VAR
VAR
	FilterWheelAxis:	FB_Axis2;
	// axis position to set to with `MoveAxis`
	position:			LREAL;
	// current filter determined from the axis position
	actual_filter:		WORD;
	FilterWheelEvent:	FB_EventLog;
	CalibratedEvent:	FB_EventLog;
	FilterReadyEvent:	FB_Eventlog;
	// last known filter position
	last_filter_position:	WORD;
END_VAR
VAR CONSTANT
	// total number of filters in the filter wheel
	filters:			WORD := 24;
	// current position of the calibration cam. Apply an offset here if necessary
	calibration_position:	LREAL := 0.0;
END_VAR

(* This program controls the filter wheel. 
The current optical filter is selected through `filter_position`.
The number of filters is hard coded to 24.

*)

// limit desired filter_position to [0...filters-1]
filter_position := filter_position MOD filters;
// calculate the actual filter position
actual_filter := LREAL_TO_WORD((360.0 - act_position) * filters / 360.0) MOD filters;

Ready := (filter_position = actual_filter) AND FilterWheelAxis.Standstill;

// TODO: Enable only on filter change
IF Enable THEN
	IF FilterWheelAxis.Calibrated THEN
		HomeAxis := FALSE;
		// if we are on automatic mode then position the filterwheel
		position := MODABS(360.0 - 360.0 * WORD_TO_LREAL(filter_position) / WORD_TO_LREAL(filters), 360.0);
		MoveAxis := filter_position <> actual_filter AND FilterWheelAxis.Standstill;
	ELSE
		position := calibration_position;
		IF FilterWheelAxis.Ready THEN
			HomeAxis := TRUE;
		END_IF
	END_IF
END_IF

Calibrated := FilterWheelAxis.Calibrated;

FilterWheelAxis(
	Enable := 			Enable,
	Reset := 			Reset,
	MoveAxis :=			MoveAxis,
	HomeAxis :=			HomeAxis,
	Position := 		position, 
	Velocity :=			60.0,
	Enable_Positive :=  TRUE,
	Enable_Negative := 	TRUE,
	Jog_Forward :=		left,
	Jog_Backwards := 	right,
	bCalibrationCam :=	NOT GVL_FilterWheel.bCalibrationCam,
	isModuloAxis :=		TRUE,
	ActualPosition => 	act_position,
	Error => 			error,
	ErrorID => 			ErrorID,
	AxisRef :=			GVL_FilterWheel.FilterWheel_AxisRef);

IF FilterWheelAxis.MoveDone THEN
	MoveAxis := FALSE;
END_IF

IF FilterWheelAxis.HomeDone THEN
	HomeAxis := FALSE;
END_IF
	
IF FilterWheelAxis.ResetDone THEN
	reset := FALSE;
END_IF

IF actual_filter <> last_filter_position THEN
	MAIN.MQTTClient.Publish('telescope', 'dome', 'FilterPosition', WORD_TO_STRING(actual_filter));
	last_filter_position := actual_filter;
END_IF

FilterWheelEvent(	
	Trigger := 		Error, 
	Level := 		ADSLOG_MSGTYPE_ERROR,
	FormatString :=	'Filter Wheel Axis Error: %s',
	OnMessage := 	NCError_TO_STRING(ErrorID),
	OffMEssage := 	'OK',
	OffLevel := 	ADSLOG_MSGTYPE_HINT);
	
CalibratedEvent(
	Trigger :=		Calibrated,
	Level := 		ADSLOG_MSGTYPE_HINT,
	FormatString :=	'%s',
	OnMessage := 	'Filter wheel is calibrated.');
	
FilterReadyEvent(
	Trigger :=		(filter_position = actual_filter),
	Level := 		ADSLOG_MSGTYPE_HINT,
	FormatString :=	'Filter position %s is ready.',
	OnMessage := 	WORD_TO_STRING(actual_filter));

END_PROGRAM

// ---- POUs/DomeControl.TcPOU
PROGRAM DomeControl
VAR_INPUT
	// enable the dome azimuth
	enable:		BOOL := TRUE;
	// reset the dome axis after an error
	Reset:		BOOL;
	// rotate the dome left (ccw)
	left:		BOOL;
	// rotate the dome right (cw)
	right: 		BOOL;
	// open the dome
	OpenDome:	BOOL;
	// close the dome
	CloseDome:	BOOL; // := TRUE;
	// turn on the light in the dome
	Light: 		BOOL;
	// azimuth position to move to
	position:	LREAL;
	// initiate homing
	HomeAxis:	BOOL;
	// rotation velocity
	velocity:	LREAL := 100.0;
END_VAR
VAR_OUTPUT
	// error condition on the azimuth drive
	Error:		BOOL;
	// NC axis error of the dome drive
	ErrorID:	UDINT;
	// error in the dome communication or drive
	DomeError:	BOOL;
	// dome is calibrated
	Calibrated:	BOOL;
END_VAR
VAR
	// dome axis function block
	DomeAxis: FB_Axis2;
	// current measured dome azimuth
	Azimuth_current: 	LREAL;
	// dome velocity
	ActVelo:			LREAL;
	//
	//manual_enable:		BOOL;
	// command to move the azimuth to position
	move_azimuth:		BOOL;
	// dome is halted
	//stop_done:			BOOL;
	// dome slit and flap are open
	DomeOpened:			BOOL;
	// dome is closed
	DomeClosed:			BOOL;
	// dome flap (lower section) is open
	FlapOpen:			BOOL;
	// dome flap (lower section) is closed
	FlapClosed:			BOOL;
	//dome slit is open
	SlitOpen:			BOOL;
	// dome slit is closed
	SlitClosed:			BOOL;
	// bit to indicate if domestatus is valid
	DomeValid:			BOOL;
	// dome control word
   	DomeStatusWord:		WORD;
	// last status Word
	LastStatus:			WORD;
	// permanent communication error
	PermanentError:		TON := (IN:=FALSE, PT:=T#30S);
	HomeDelay:			FB_TONTP;
	F_Azimuth_home:		F_TRIG;
	R_Azimuth_home:		R_TRIG;
	// direction invariant azimuth home signal;
	Azimuth_home:		BOOL;
	// time delay for dome light
	LightTimer:			TP;
	// next state
	//:				BYTE := 0;
	// ADS communiaction busy
	bBusy: 				BOOL;
	// ADS communication error
	bError: 			BOOL;
	// ADS communication error id
	nErrID: 			UDINT;
	// cycle timer for the ADS write cycle
	ReadCycle:			TON := (PT:=T#1S);
	
	fbReadReq: ADSREAD := ( NETID := '5.73.45.158.1.1', PORT := 851, TMOUT := DEFAULT_ADS_TIMEOUT );
	DomeCalibration:	MC_SetPosition;
	HomingMode:			MC_HomingMode := MC_DefaultHoming;
	SyncDome:			BOOL;
	DomeCommEvent:		FB_Eventlog;
	DomeAxisEvent:		FB_Eventlog;
	DomeOpenedEvent:	FB_Eventlog;
	DomeClosedEvent:	FB_Eventlog;
	OpenDomeEvent:		FB_Eventlog;
	CloseDomeEvent:		FB_Eventlog;
	DomeCalibrationEvent: FB_Eventlog;
	MQTTTimer : TON := (PT:=T#10S);
	getlastposition:	BOOL := TRUE;
END_VAR
VAR CONSTANT
	tolerance:				LREAL := 5.0;
	calibration_position:	LREAL := 172.5;
//	home_position:			LREAL := 180.0;
END_VAR
VAR PERSISTENT
	last_position:	LREAL := -1.0;
END_VAR

(* This program is responsible for the dome control. 
The dome is enabled unless the emergency button is pressed.
The two-button manual box steers the dome counter-clockwise or clockwise
If the dome is in automatic mode, homing is performed first.
The first section controls the signals for the inverter.
The second section controls the dome axis.
The third section handles the communications via ADS with the dome PLC.
*)

DomeLowLevelControl(enable := GVL_Safety.Run);

// if we are calibrated or encounter an error while calibrating, deactivate homing
IF DomeAxis.Calibrated OR Error THEN
	HomeAxis := FALSE;
END_IF

IF Error THEN
	move_azimuth := FALSE;
END_IF

IF DomeAxis.Calibrated THEN
	last_position := Azimuth_current;
	getlastposition := FALSE;
END_IF


ActVelo := GVL_Dome.ActVelo;

// limit position to sane value
position := MODABS(position, 360.0);

// if we are calibrated, but azimuth is not, go to home position
HomeDelay(IN := DomeAxis.Calibrated, PT1 := T#5S, PT2 := T#100MS);
(*
IF HomeDelay.Q THEN
	position := home_position;
	move_azimuth := TRUE;
END_IF
*)
SyncDome := DomeAxis.Calibrated AND TelescopeControl.ready AND TelescopeControl.telescope_mode = E_TelescopeMode.automatic;
// if we are on automatic, tie the dome to the telescope

IF SyncDome THEN
	position := MODABS(TelescopeControl.azimuth_current, 360.0);
	IF ABS(Azimuth_current - position) > tolerance THEN
		velocity := 100.0;
		move_azimuth := TRUE;
	ELSE
		move_azimuth := FALSE;
	END_IF
	
END_IF

IF DomeClosed AND Calibrated AND TelescopeControl.telescope_mode = E_TelescopeMode.automatic THEN
	IF Environment.WindSpeed > 10.0 THEN
		position := Environment.WindDirection;
		move_azimuth := TRUE;
	ELSE
		move_azimuth := FALSE;
	END_IF
END_IF

Calibrated := DomeAxis.Calibrated;
// automaticallz calibrate dome
IF TelescopeControl.telescope_mode = E_TelescopeMode.automatic AND enable THEN
	HomeAxis := NOT Calibrated;
END_IF

F_Azimuth_home(CLK := GVL_Dome.Azimuth_home);
R_Azimuth_home(CLK := GVL_Dome.Azimuth_home);

Azimuth_home := (R_Azimuth_home.Q AND GVL_Dome.bDirectionPlus) OR 
				(F_Azimuth_home.Q AND GVL_Dome.bDirectionMinus) OR
				(GVL_Dome.Azimuth_home AND DomeAxis.StandStill);

				// when homing, ensure that the position is the calibration position
IF HomeAxis THEN
	IF last_position > 0.0 THEN // direct calibration
		HomingMode := MC_ForceCalibration; // MC_Direct
		DomeCalibration.Position := last_position;
		DomeCalibration.Execute := TRUE;
	ELSE // classic calibration
		HomingMode := MC_DefaultHoming;
		position := calibration_position;
		// set to slow velocity for homing
		velocity := 15.0;
		DomeCalibration.Execute := FALSE;
	END_IF
ELSE // we are not homing
	velocity := 100.0;
	DomeCalibration.Execute := FALSE;	
END_IF


IF Calibrated AND Azimuth_home THEN
	DomeCalibration.Position := calibration_position;
	DomeCalibration.Execute := TRUE;
END_IF

// velocity = 2°/s or 180° in 81s, 360° in 120s (was 2.22)
// TODO: Reset does not propagate to the FB and therefor does not reset the error
DomeAxis(
	Enable := 		enable AND GVL_Safety.Run,
	Reset := 		reset,
	MoveAxis := 	move_azimuth,
	HomeAxis :=		HomeAxis,
	HomingMode :=	HomingMode,
	Position := 	position,
	Velocity := 	velocity,
	Jog_Forward :=	right OR GVL_Dome.Clockwise,
	Jog_Backwards := left OR GVL_Dome.CounterClockwise,
	bCalibrationCam := GVL_Dome.Azimuth_home,
	isModuloAxis := TRUE,
	//StopDone =>		stop_done,
	Error =>		error,
	ErrorID =>		ErrorID,
	ActualPosition => Azimuth_current,
	AxisRef	:= 		GVL_Dome.DomeAxisRef);



// re-calibrate the dome, if we pass the reference switch. execute only if enough time has passed since homing.
DomeCalibration(Axis := GVL_Dome.DomeAxisRef);

IF DomeCalibration.Done OR Calibrated THEN
	getlastposition := FALSE;
END_IF
(*
IF DomeAxis.MoveDone THEN
	move_azimuth := FALSE;
END_IF
*)

// Light is switched off after 60 minutes or if Light signal is low
LightTimer(IN := Light, PT := T#60M);
GVL_Dome.Light := Light AND LightTimer.Q;

(* The remote section for moving parts of the dome starts here. *)
GVL_Dome.DomeControlWord.0 := TRUE;
IF CloseDome THEN
	OpenDome := FALSE;
	GVL_Dome.DomeControlWord.1 := TRUE; // CloseFlap
	GVL_Dome.DomeControlWord.2 := TRUE; // CloseSlit
	GVL_Dome.DomeControlWord.3 := FALSE; // OpenFlap
	GVL_Dome.DomeControlWord.4 := FALSE; // OpenSlit
ELSIF OpenDome THEN
	GVL_Dome.DomeControlWord.1 := FALSE; // CloseFlap
	GVL_Dome.DomeControlWord.2 := FALSE; // CloseSlit
	GVL_Dome.DomeControlWord.3 := TRUE; // OpenFlap
	GVL_Dome.DomeControlWord.4 := TRUE; // OpenSlit
ELSE
	GVL_Dome.DomeControlWord.1 := FALSE; // CloseFlap
	GVL_Dome.DomeControlWord.2 := FALSE; // CloseSlit
	GVL_Dome.DomeControlWord.3 := FALSE; // OpenFlap
	GVL_Dome.DomeControlWord.4 := FALSE; // OpenSlit
END_IF

ReadCycle(IN := TRUE);
IF ReadCycle.Q THEN
	// read if the ADS command is busy
	fbReadReq(	READ := FALSE,
				BUSY => bBusy,
				ERR =>	bError);
	IF bBusy THEN
		// reset the read command
		fbReadReq(READ := FALSE);
	ELSE
		// read the variable
		fbReadReq(  IDXGRP := 16#4020, 
					IDXOFFS := 0, 
					LEN := SIZEOF(DomeStatusWord), 
					DESTADDR := ADR(DomeStatusWord),
					READ := TRUE,
					BUSY => bBusy,
					ERR =>	bError);
		// restart the read cycle
		ReadCycle(IN := FALSE);		
	END_IF
	
	IF NOT bError THEN
		DomeValid  := DomeStatusWord.0;
		DomeOpened := DomeStatusWord.1;
		DomeClosed := DomeStatusWord.2;
		FlapOpen   := DomeStatusWord.3;
		FlapClosed := DomeStatusWord.4;
		SlitOpen   := DomeStatusWord.5;
		SlitClosed := DomeStatusWord.6;
	ELSE
		// reset the status word
		nErrID := fbReadReq.ERRID;
		DomeStatusWord := 0;
	END_IF
END_IF

CASE NErrID OF
			6: DomeCommEvent.OnMessage := 'ERR_TARGETPORTNOTFOUND';
			29: DomeCommEvent.OnMessage := 'ERR_AMSSYNC_TIMEOUT';
			1861: DomeCommEvent.OnMessage := 'ADSERR_CLIENT_SYNCTIMEOUT';
ELSE
			DomeCommEvent.OnMessage := UDINT_TO_STRING(nErrID);
END_CASE

PermanentError(IN := NOT DomeValid);
		
DomeError := PermanentError.Q OR Error;

IF DomeOpened THEN
	OpenDome := FALSE;
ELSIF DomeClosed THEN
	CloseDome := FALSE;
END_IF

MQTTTimer(IN:=Enable);
IF MQTTTimer.Q THEN // publish new payload every second
	MQTTTimer(IN:=FALSE);
	MAIN.MQTTClient.Publish('dome', 'dome', 'DomeAzimuth', LREAL_TO_FMTSTR(Azimuth_current, 1, TRUE));
	MAIN.MQTTClient.Publish('dome', 'dome', 'DomeCalibrated', BOOL_TO_STRING(Calibrated));	
	// invalidate last status for testing
	LastStatus := 0;
END_IF

IF DomeStatusWord <> LastStatus THEN
	LastStatus := DomeStatusWord;
	MAIN.MQTTClient.Publish('dome', 'dome', 'DomeCommunicationOK', BOOL_TO_STRING(NOT PermanentError.Q));
	MAIN.MQTTClient.Publish('dome', 'dome', 'DomeClosed', BOOL_TO_STRING(DomeClosed));
	MAIN.MQTTClient.Publish('dome', 'dome', 'DomeOpened', BOOL_TO_STRING(DomeOpened));
	MAIN.MQTTClient.Publish('dome', 'dome', 'FlapOpen', BOOL_TO_STRING(FlapOpen));	
	MAIN.MQTTClient.Publish('dome', 'dome', 'FlapClosed', BOOL_TO_STRING(FlapClosed));	
	MAIN.MQTTClient.Publish('dome', 'dome', 'SlitOpen', BOOL_TO_STRING(SlitOpen));	
	MAIN.MQTTClient.Publish('dome', 'dome', 'SlitClosed', BOOL_TO_STRING(SlitClosed));	
END_IF

DomeCommEvent(	Trigger := PermanentError.Q, 
					Level := ADSLOG_MSGTYPE_ERROR,
					FormatString := 'Dome communication error: %s',
					OffMessage := 'OK',
					OffLevel := ADSLOG_MSGTYPE_HINT);
DomeAxisEvent(	
	Trigger := 		Error, 
	Level := 		ADSLOG_MSGTYPE_ERROR,
	FormatString :=	'Dome axis Error: %s',
	OnMessage := 	NCError_TO_STRING(ErrorID),
	OffMEssage := 	'OK');
				
DomeCalibrationEvent(	
	Trigger := 		GVL_Dome.Azimuth_home, 
	Level := 		ADSLOG_MSGTYPE_HINT,
	OnMessage := 	'Dome is (re-)calibrated.');

DomeOpenedEvent(
	Trigger := 		DomeOpened, 
	Level := 		ADSLOG_MSGTYPE_WARN,
	OnMessage := 	'Dome is open.');
	
DomeClosedEvent(
	Trigger := 		DomeClosed, 
	Level := 		ADSLOG_MSGTYPE_HINT,
	OnMessage := 	'Dome is closed.');
	
OpenDomeEvent(
	Trigger := 		OpenDome, 
	Level := 		ADSLOG_MSGTYPE_WARN,
	OnMessage := 	'Dome is opening.');
	
CloseDomeEvent(
	Trigger := 		CloseDome, 
	Level := 		ADSLOG_MSGTYPE_HINT,
	OnMessage := 	'Dome is closing.');

END_PROGRAM

// ---- POUs/DomeLowLevelControl.TcPOU
PROGRAM DomeLowLevelControl
VAR_INPUT
	enable : BOOL;
END_VAR
VAR
	Inverter_Enable:	BOOL;
	Inverter_Velocity:	UINT;
END_VAR

(* source: https://infosys.beckhoff.de/english.php?content=../content/1033/tcplclib_tc2_system/18014399220202635.html&id= *)

IF GVL_Dome.bVeloHigh THEN
	// High Speed
	Inverter_Velocity := 32767;
	Inverter_Enable := enable;
ELSIF GVL_Dome.bVeloLow THEN
	// low speed
	Inverter_Velocity := 10000;
	Inverter_Enable := enable;
ELSIF GVL_Dome.bBreak THEN
	// breaking (halt)
	Inverter_Velocity := 0;
	Inverter_Enable := FALSE;
ELSE
	// default
	Inverter_Velocity := 0;
	Inverter_Enable := FALSE;
END_IF

GVL_Dome.Inverter_DirectionMinus := GVL_Dome.bDirectionPlus;
GVL_Dome.Inverter_Enable := Inverter_Enable;
GVL_Dome.Inverter_Velocity := Inverter_Velocity;

END_PROGRAM

// ---- POUs/Environment.TcPOU
PROGRAM Environment
VAR_OUTPUT
	// wind speed in m/s
	WindSpeed:		REAL;
	// wind direction in degrees
	WindDirection:	REAL;
	// outside temperature in degrees celsius
	Temperature:	REAL;
	// humidity in percent (0...100)
	Humidity:		REAL;
	// Pressure in mBars
	Pressure:		REAL;
	// Brightness in lux
	Brightness:		REAL;
	// incoming light direction (solar azimuth)
	LightDirection:	REAL;
	// rain in mm/h
	Precipitation:	REAL;
	// dome temperature in degrees
	TemperatureDome:REAL;
	// dome humidity in percent
	HumidityDome:	REAL;
	// dome dewpoint in degrees celsius
	DewpointDome:	REAL;
	// boolean rain event
	Rain:			BOOL;
	// boolean weather bad condition
	WeatherBad:		BOOL;
	// boolean weather good condition for observation
	WeatherGood:	BOOL;
END_VAR
VAR
	WindEvent,
	HumidityEvent,
	HumidityDomeEvent,
	PrecipitationEvent,
	DewpointEvent,
	WeatherGoodEvent: FB_Eventlog;
	WindAverage,
	Wind5sAverage,
	WindDirectionAverage,
	HumidityDomeAverage,
	PressureAverage,
	PrecipitationAverage,
	BrightnessAverage: FB_TimeAverage;
	RainDelay:	TON;
	RainSustain: TOF;
	sunpos:		FB_SUNPOS;
	eq2hor2:	FB_EQ2HOR2;
	avg_wind, max_wind: REAL;
	HumidityThreshold:	SR;
	HumidityDomeThreshold:	SR;
	WindThreshold:		SR;
	WeatherBadDelay: 	TOF;
	MQTTTimer : TON := (PT:=T#10S);
END_VAR

(* convert raw Sensor values to real values 
calibration values in Thiess Clima manual table 9*)
WindSpeed := 		F_YREAL(GVL_Environment.rawWindSpeed, 		0, 32767,   0.0, 60.0); // m/s
WindDirection :=	F_YREAL(GVL_Environment.rawWindDirection, 	0, 32767,   0.0, 360.0); // °
Temperature :=  	F_YREAL(GVL_Environment.rawTemperature, 	0, 32767, -40.0, 60.0); // °C -40...80?
Humidity :=			F_YREAL(GVL_Environment.rawHumidity, 		0, 32767,   0.0, 100.0); // %
Pressure := 		F_YREAL(GVL_Environment.rawPressure,		0, 32767, 800.0, 1060.0); // mBar 
Brightness := 		F_YREAL(GVL_Environment.rawBrightness,		0, 32767,   0.0, 120000.0); // Lux 
LightDirection :=	F_YREAL(GVL_Environment.rawLightDirection, 	0, 32767,   0.0, 360.0); // °
Precipitation := 	F_YREAL(GVL_Environment.rawPrecipitation - 28,	0, 32767,   0.0, 100.0); // mm/h 
HumidityDome :=		F_YREAL(GVL_Environment.rawHumidityDome, 		0, 32767,   0.0, 100.0); // %
TemperatureDome :=  F_YREAL(GVL_Environment.rawTemperatureDome, 	0, 32767, -30.0, 70.0); // °C

DewpointDome := 	F_Dewpoint(HumidityDome, TemperatureDome);

RainDelay(IN := GVL_Environment.rawRain OR NOT GVL_Environment.rawNoRain, PT := T#60S);
RainSustain( IN := RainDelay.Q, PT := T#120S, Q => Rain);
WindAverage(IN := WindSpeed, PT := T#3M, AVG => avg_wind, MAXAVG => max_wind);
Wind5sAverage(IN := WindSpeed, PT := T#10S);
WindDirectionAverage(IN := WindDirection, PT := T#5S);
PressureAverage(IN := Pressure, PT := T#5S);
PrecipitationAverage(IN := Precipitation, PT := T#60S);
BrightnessAverage(IN := Brightness, PT := T#10S);

// addition rules for low values
IF Brightness < 250.0 THEN
	Brightness := BrightnessAverage.AVG;
END_IF
// Thresholds
HumidityThreshold(	SET1 := Humidity >= 80.0,
					RESET := Humidity < 65.0);

HumidityDomeThreshold(	SET1 := HumidityDome >= 80.0,
					RESET := HumidityDome <= 65.0);

WindThreshold(	SET1 := WindAverage.AVG > 10.0 OR max_wind > 15.0, 
				RESET := WindAverage.AVG < 5.0);

WeatherBadDelay(IN := Rain OR
				PrecipitationAverage.AVG >= 0.1 OR
				HumidityThreshold.Q1 OR
				HumidityDomeThreshold.Q1 OR
				WindThreshold.Q1, PT := T#4M, Q => WeatherBad);
// close dome on bad weather				
IF WeatherBad AND DomeControl.DomeOpened THEN
	DomeControl.CloseDome := TRUE;
END_IF

// calculate solar position
sunpos(JD := TelescopeControl.jd);
eq2hor2(alpha := sunpos.RA,
	delta := sunpos.Dec,
	lon := TelescopeControl.longitude,
	lat := TelescopeControl.latitude,
	JD := TelescopeControl.jd);

WeatherGood := NOT WeatherBad AND eq2hor2.alt<0.0;
	
MQTTTimer(IN:=TRUE);
IF MQTTTimer.Q THEN // publish new payload every second
	MQTTTimer(IN:=FALSE);
	MAIN.MQTTClient.Publish('environment', 'roof', 'OutsideTemperature', LREAL_TO_FMTSTR(Temperature, 2, TRUE));
	MAIN.MQTTClient.Publish('environment', 'roof', 'OutsideHumidity', LREAL_TO_FMTSTR(Humidity, 1, TRUE));
	MAIN.MQTTClient.Publish('environment', 'roof', 'WindSpeed', LREAL_TO_FMTSTR(Wind5sAverage.AVG, 1, TRUE));
	MAIN.MQTTClient.Publish('environment', 'roof', 'WindSpeedMax', LREAL_TO_FMTSTR(Wind5sAverage.MAXAVG, 1, TRUE));
	MAIN.MQTTClient.Publish('environment', 'roof', 'WindDirection', LREAL_TO_FMTSTR(WindDirectionAverage.AVG, 1, TRUE));
	MAIN.MQTTClient.Publish('environment', 'roof', 'Pressure', LREAL_TO_FMTSTR(PressureAverage.AVG, 2, TRUE));
	MAIN.MQTTClient.Publish('environment', 'roof', 'Brightness', LREAL_TO_FMTSTR(Brightness, 2, TRUE));
	MAIN.MQTTClient.Publish('environment', 'roof', 'LightDirection', LREAL_TO_FMTSTR(LightDirection, 1, TRUE));
	MAIN.MQTTClient.Publish('environment', 'roof', 'Rain', BOOL_TO_STRING(Rain));
	MAIN.MQTTClient.Publish('environment', 'roof', 'RainAnalog', LREAL_TO_FMTSTR(PrecipitationAverage.AVG, 3, TRUE));
	MAIN.MQTTClient.Publish('environment', 'roof', 'solz', LREAL_TO_FMTSTR(90.0 - eq2hor2.alt, 3, TRUE));
	MAIN.MQTTClient.Publish('environment', 'roof', 'solaz', LREAL_TO_FMTSTR(eq2hor2.az, 3, TRUE));
					
	MAIN.MQTTClient.Publish('dome', 'dome', 'DomeTemperature', LREAL_TO_FMTSTR(TemperatureDome, 2, TRUE));
	MAIN.MQTTClient.Publish('dome', 'dome', 'DomeHumidity', LREAL_TO_FMTSTR(HumidityDome, 1, TRUE));
	MAIN.MQTTClient.Publish('dome', 'dome', 'WeatherBad', BOOL_TO_STRING(WeatherBad));
	MAIN.MQTTClient.Publish('dome', 'dome', 'WeatherGood', BOOL_TO_STRING(WeatherGood));
END_IF

WindEvent(	Trigger := avg_wind > 10.0, 
			Level := ADSLOG_MSGTYPE_WARN,
			FormatString := 'Wind Speed: %s',
			OnMessage := LREAL_TO_FMTSTR(WindSpeed, 2, TRUE),
			OffMessage := 'OK',
			OffLevel := ADSLOG_MSGTYPE_HINT);

HumidityEvent(	Trigger :=  HumidityThreshold.Q1 AND DomeControl.DomeOpened, 
				Level := ADSLOG_MSGTYPE_WARN,
				FormatString := 'Humidity: %s',
				OnMessage := LREAL_TO_FMTSTR( Humidity, 1, TRUE),
				OffMessage := 'OK',
				OffLevel := ADSLOG_MSGTYPE_HINT);

// azimuth encoder starts to fail at 65% humidity
HumidityDomeEvent(	Trigger :=  HumidityDomeAverage.AVG>= 65.0, 
				Level := ADSLOG_MSGTYPE_WARN,
				FormatString := 'Humidity in Dome: %s',
				OnMessage := LREAL_TO_FMTSTR( HumidityDomeAverage.AVG, 1, TRUE),
				OffMessage := 'OK',
				OffLevel := ADSLOG_MSGTYPE_HINT);

				
PrecipitationEvent(	Trigger := WeatherBad AND DomeControl.DomeOpened, 
					Level := ADSLOG_MSGTYPE_WARN,
					FormatString := 'The weather is %s',
					OnMessage := 'BAD.',
					OffMessage := 'OK.');

WeatherGoodEvent(	Trigger := WeatherGood, 
					Level := ADSLOG_MSGTYPE_HINT,
					FormatString := 'The weather is %s',
					OnMessage := 'good: virtual dome is open.',
					OffMessage := 'bad: virtual dome is closed.',
					OffLevel := ADSLOG_MSGTYPE_HINT);


DewPointEvent( Trigger := TemperatureDome < DewpointDome,
				Level := ADSLOG_MSGTYPE_WARN,
				FormatString := 'Dewpoint in Dome below ambient Temperature: %s',
				OnMessage := LREAL_TO_FMTSTR( DewpointDome, 1, TRUE),
				OffMessage := 'OK',
				OffLevel := ADSLOG_MSGTYPE_HINT);

END_PROGRAM

// ---- POUs/FunctionBlocks/FB_TimeAverage.TcPOU
FUNCTION_BLOCK FB_TimeAverage
VAR_INPUT
	IN:		REAL;
	PT:		TIME := T#4400MS;
END_VAR
VAR_OUTPUT
	AVG:	REAL;
	MINAVG:	REAL;
	MAXAVG:	REAL;
	Overflow: BOOL;
END_VAR
VAR
	fbCycle	:TON;
	buffer:	ARRAY[0..30000] OF REAL;
	index:	INT := 0;
	number:	INT := 0;
	i:		INT;
	sum:	REAL;
END_VAR

fbCycle(IN:= NOT fbCycle.Q,
		PT:= PT);

// write the current value into the buffer		
buffer[index] := IN;

// increase the index
IF index < 30000 THEN
	index := index + 1;
END_IF

Overflow := (index = 30000);

// during the first cycle number will be smaller than index
IF number < index THEN
	number := index;
END_IF

// sum up the buffer to the current number
sum := 0.0;
MINAVG := IN;
MAXAVG := IN;
FOR i :=0 TO number-1 DO
	sum := sum + buffer[i];
	MINAVG := MIN(buffer[i], MINAVG);
	MAXAVG := MAX(buffer[i], MAXAVG);
END_FOR

// return the average
AVG := sum / number;

// if we hit the cycle time, reset the index and overwrite old values
IF fbCycle.Q THEN
	number := index;
	index := 0;
END_IF

END_FUNCTION_BLOCK

// ---- POUs/Functions/F_YREAL.TcPOU
FUNCTION F_YREAL : REAL
VAR_INPUT
	fX:		LREAL;
	fXmin:	REAL := 0.0;
	fXmax:	REAL := 32767.0;
	fYmin:	REAL := 0.0;
	fYmax:	REAL := 1.0;
END_VAR
VAR
	fgain:		LREAL;
	foffset:	LREAL;
END_VAR

(*
y = mx+b

		    delta X	  fYmax - fYmin
m = fgain = ------- = -------------
			delta Y	  fXmax - fXmin
			
b = foffset = y - m*x = y - fgain*x
					  = fYmin - fgain * fXmin
*)

// y = fgain * x + foffset

IF (fXmax - fXmin) <> 0 THEN

	// Berechnung der Steigung
	fgain := (fYmax - fYmin) / (fXmax - fXmin);
	
	// Berechnung des Offsets
	foffset := fYmin - (fgain * fXmin);
	
	// Berechnung von F_Y

	F_YREAL := LREAL_TO_REAL(fgain * fX + foffset);
	F_YREAL := LIMIT(fYmin, F_YREAL, fYMAX);
END_IF

END_FUNCTION

// ---- POUs/Functions/F_Dewpoint.TcPOU
FUNCTION F_Dewpoint : REAL
VAR_INPUT
	// relative humidity
	relhum:	REAL;
	// temperature °C
	t: REAL;
END_VAR
VAR
	a, b, 
	// Sättigungsdampfdruck in hPa
	sdd, 
	// Dampfdruck in hPa
	dd, v: REAL;
END_VAR

// source https://www.wetterochs.de/wetter/feuchte.html
IF t < 0.0 THEN
	a := 7.6; b := 240.7;// für T < 0 über Wasser (Taupunkt)
ELSE
	a := 7.5; b := 237.3;
END_IF

F_Dewpoint := -273.15;
IF b+T > 0.0 THEN
	SDD := LREAL_TO_REAL(6.1078 * EXPT(10, (a*T)/(b+T)));
ELSE
	SDD := 6.1078;
END_IF

IF SDD > 0.0 THEN
	DD := relhum/100.0 * SDD;
END_IF

IF DD  > 0.0 THEN
  v := LOG(ABS(DD)/6.1078);	
END_IF

IF a <> v THEN
	F_Dewpoint := b*v/(a-v);	
END_IF

END_FUNCTION

// ---- POUs/FocusControl.TcPOU
PROGRAM FocusControl
VAR_INPUT
	// enable the axis
	enable: BOOL;
	// Move M2 closer to M1
	inward: 	BOOL;
	// Move M2 away from M1
	outward: 	BOOL;	
	// reset the axis(-error)
	reset: 		BOOL;
	// move the axis to new position
	MoveAxis:	BOOL;
	// calibrate the focus axis
	HomeAxis:	BOOL;
	// focus position in millimeters
	position: 		LREAL;
END_VAR

VAR_OUTPUT
	// true if absolute calibration
	Calibrated:	BOOL;
	// true if error
	Error: 		BOOL;
	// ID of NC axis error
	ErrorID:	UDINT;
	// ready signal = drive ready + standstill
	Ready:	BOOL;
END_VAR

VAR
	FocusDelay:			TON;
	BrakeDelay:			TON;
	FocusAxis:			FB_Axis2;
	actual_position:	LREAL;
	FocusUnlock:		BOOL;
	FocusUnlocked:		BOOL;
	SetPosition:		MC_SetPosition;
	HomingMode:			MC_HomingMode := MC_DefaultHoming;
	MQTTTimer : 		TON := (PT:=T#5S);
	FocusAxisEvent:		FB_EventLog;
	CalibrationEvent:	FB_EventLog;
END_VAR

VAR CONSTANT
	// reference position for homing
	homing_position:		LREAL := 97.96; // 107,50 - 9,54
	//calibration_position:	LREAL := 0.0;
	tolerance:				LREAL := 0.005;
END_VAR
VAR PERSISTENT
	last_position:	LREAL := -1.0;
END_VAR

(*
Focus Control Unit
spindle gear: 5mm
brake: 86 61103H00 Var. 0005 Index C; 24VDC geglattet 0,25 A P1672/R7
motor: Faulhaber ; Schönaich ; 3557K024CR; 454  431 ; Made in germany ==> 5300 rpm
gear: Faulhaber ; MINIMOTOR SA ; swiss made ; 38/1S  43:1 ; 033896  503
Focus is locked by default
*)

GVL_Telescope.focus_unlock := FocusUnlock OR enable;

// wait until the focus is unlocked for n milliseconds
FocusDelay(IN := GVL_Telescope.focus_unlock, PT := T#500MS, Q => FocusUnlocked);
// wait for brake until we are at rest
BrakeDelay(IN := NOT FocusAxis.Busy AND FocusAxis.StandStill, PT := T#4000MS);

// if we are on automatic mode then position the filterwheel
IF Telescopecontrol.telescope_mode = E_TelescopeMode.automatic AND NOT FocusUnlock THEN
	IF FocusAxis.Calibrated THEN
		IF ABS(position - actual_position) > tolerance THEN
			IF FocusAxis.Ready THEN
				MoveAxis := TRUE;
			ELSE
				Enable := TRUE;
			END_IF
		END_IF
		// disable the drive and lock the brake, if we stand for more than n seconds
		IF BrakeDelay.Q THEN
			Enable := FALSE;
		END_IF
		// store actual position, if we are calibrated and locked
		IF NOT GVL_Telescope.focus_unlock THEN
			last_position := actual_position;
		END_IF
	ELSE // not calibrated
		IF FocusAxis.Ready THEN
			HomeAxis := TRUE;
		END_IF
	END_IF
END_IF

IF HomeAxis THEN
	IF last_position > 0.0 THEN
		HomingMode := MC_ForceCalibration; // MC_Direct
		position := last_position;
		SetPosition.Execute := TRUE;
	ELSE
		HomingMode := MC_DefaultHoming;
		position := homing_position;
		SetPosition.Execute := FALSE;
	END_IF
ELSE
	SetPosition.Execute := FALSE;	
END_IF

// deactivate limit switches on homing
MC_SetAcceptBlockedDriveSignal(
	Axis := GVL_Telescope.FocusAxisRef, 
	Enable := HomeAxis);

SetPosition(
	Axis := GVL_Telescope.FocusAxisRef, 
	Position := last_position);
	
FocusAxis(	
	Enable := 			FocusUnlocked,
	Reset := 			reset,
	MoveAxis := 		MoveAxis AND FocusUnlocked,
	HomeAxis :=			HomeAxis AND FocusUnlocked,
	HomingMode :=		HomingMode,
	Position := 		position,
	Velocity :=			5.0,
	Enable_Positive := 	NOT GVL_Telescope.focus_limit_far OR HomeAxis,
	Enable_Negative := 	NOT GVL_Telescope.focus_limit_near,
	Jog_Forward :=		outward AND FocusUnlocked,
	Jog_Backwards := 	inward AND FocusUnlocked,
	bCalibrationCam :=  GVL_Telescope.focus_limit_far,
	ActualPosition => 	actual_position,
	Error =>			error,
	ErrorID =>			ErrorID,
	AxisRef :=			GVL_Telescope.FocusAxisRef);	

IF FocusAxis.MoveDone THEN
	MoveAxis := FALSE;
END_IF

IF FocusAxis.HomeDone THEN
	HomeAxis := FALSE;
	Enable := FALSE;
	last_position := position;
END_IF
	
IF FocusAxis.ResetDone THEN
	reset := FALSE;
END_IF

IF FocusAxis.Calibrated OR Error THEN
	HomeAxis := FALSE;
END_IF

IF Error THEN
	last_position := -1.0;
	//FocusAxis.Calibrated := FALSE;
	Calibrated := FALSE;
END_IF

Calibrated := FocusAxis.Calibrated;

Ready := FocusAxis.Ready AND FocusAxis.StandStill OR NOT GVL_Telescope.focus_unlock;

MQTTTimer(IN:=TRUE);
IF MQTTTimer.Q THEN // publish new payload every second
	MQTTTimer(IN:=FALSE);
	MAIN.MQTTClient.Publish('telescope', 'dome', 'FocusPosition', LREAL_TO_FMTSTR(actual_position, 5, TRUE));
	MAIN.MQTTClient.Publish('telescope', 'dome', 'FocusCalibrated', BOOL_TO_STRING(Calibrated));	
	MAIN.MQTTClient.Publish('telescope', 'dome', 'FocusReady', BOOL_TO_STRING(Ready));	
END_IF

FocusAxisEvent(	
	Trigger := 		FocusAxis.Error, 
	Level := 		ADSLOG_MSGTYPE_ERROR,
	FormatString :=	'Focus Axis Error: %s',
	OnMessage := 	NCError_TO_STRING(ErrorID),
	OffMEssage := 	'OK',
	OffLevel := 	ADSLOG_MSGTYPE_HINT);

CalibrationEvent(
	Trigger :=	Calibrated,
	Level :=	ADSLOG_MSGTYPE_HINT,
	OnMessage := 'Focus is calibrated.'
	);

END_PROGRAM

// ---- POUs/DerotatorControl.TcPOU
PROGRAM DerotatorControl
VAR_INPUT
	// enable the derotator
	enable:		BOOL;
	// reset an error
	reset:		BOOL;
	// decrease derotator angle
	left:		BOOL;
	// increase derotator angle
	right:		BOOL;
	// set the absolute position
	position:	LREAL;
	// derotator velocity
	Velocity:	LREAL := 10.0;
	// move to given position
	MoveAxis: 	BOOL;
	// calibrate the axis
	HomeAxis:	BOOL;
	// tracking flag
	Tracking:	BOOL;
END_VAR
VAR_OUTPUT
	// error flag
	Error:				BOOL;
	// nc error id
	ErrorID:			UDINT;
	// actual position of the derotator
	actual_position:	LREAL;
	// calibrated flag
	Calibrated:			BOOL;
	// axis ready flag
	Ready:				BOOL;
	// position to move the axis to
	slewtime: 			LREAL;
END_VAR
VAR
	// trigger for the torque error
	TorqueError:		TON := (PT := T#3S);
	// axis function block
	DerotatorAxis:		FB_Axis2;
	
	DerotatorEvent:		FB_EventLog;
	// torque warning event
	TorqueWarning:		FB_EventLog;
	// torque calibration event
	CalibrationEvent:	FB_EventLog;
	// percentage of the derotator torque
	derotator_torque:	REAL;
	ReadParameter:		MC_ReadParameter;
END_VAR
VAR CONSTANT
	// current position of the calibration cam. Apply an offset here if necessary
	calibration_position:	LREAL := 438.4623; // calibration in positive direction (was 460.0)
END_VAR

(*
Selection 6
Homing in Endlage:

https://infosys.beckhoff.com/index.php?content=../content/1031/ax5000_usermanual/html/ax5000_homing_hardware_end_position.htm&id=12221
NC-Interface:
PlcToNc-Achsinterface, Bit 8 namens AcceptBlockedDriveSignal im nDeCtrlDWord

SPS-Interface:
TcNc-Lib, siehe SPS-Funktion AxisSetAcceptBlockedDriveSignal in der TwinCAT  PLC Library: NC.
*)

position := LIMIT(calibration_position - 460.0, position, calibration_position);

// WARNING: Homing disables the limit Switches!

MC_SetAcceptBlockedDriveSignal(
	Axis := GVL_Telescope.DerotatorAxisRef,
	Enable := HomeAxis);


IF DerotatorAxis.Calibrated THEN
	HomeAxis := FALSE;
	Calibrated := DerotatorAxis.Calibrated;
END_IF
	
IF HomeAxis THEN
	position := calibration_position;
END_IF

IF Tracking THEN
	IF ABS(actual_position - position) > 1.0 THEN
		Tracking := FALSE;
		MoveAxis := TRUE;
	ELSE
		MoveAxis := FALSE;
	END_IF
END_IF

DeRotatorAxis(
	enable := 			enable,
	Reset := 			Reset,
	MoveAxis :=			MoveAxis,
	HomeAxis :=			HomeAxis,
	Position := 		position, 
	Velocity :=			Velocity,
	Enable_Positive := 	NOT GVL_Telescope.Derotator_inputs.0 OR HomeAxis,
	Enable_Negative := 	NOT GVL_Telescope.Derotator_inputs.1,
	Jog_Forward := 		right,
	Jog_Backwards := 	left,
	bCalibrationCam :=	GVL_Telescope.Derotator_inputs.0,
	isModuloAxis :=		FALSE,
	Tracking :=			Tracking,
	ActualPosition => 	actual_position,
	Error => 			Error,
	ErrorID => 			ErrorID,
	AxisRef :=			GVL_Telescope.DerotatorAxisRef);
	
IF DeRotatorAxis.MoveDone OR Reset OR Error THEN
	MoveAxis := FALSE;
END_IF

IF DeRotatorAxis.HomeDone OR Reset OR Error THEN
	HomeAxis := FALSE;
END_IF
	
IF DeRotatorAxis.ResetDone THEN
	reset := FALSE;
END_IF

Ready := DeRotatorAxis.Ready;

ReadParameter(	Axis := GVL_Telescope.DerotatorAxisRef, 
				Enable := DeRotatorAxis.InMotion, 
				ParameterNumber := MC_AxisParameter.AxisRemainingTimeToGo, 
				ReadMode := E_ReadMode.READMODE_CYCLIC);
				
IF ReadParameter.Valid THEN
	slewtime := ReadParameter.Value;
END_IF

derotator_torque := GVL_Telescope.Derotator_torque / 10.0;

TorqueError(IN := ABS(derotator_torque) > 16.0);

DerotatorEvent(	
	Trigger := 		Error, 
	Level := 		ADSLOG_MSGTYPE_ERROR,
	FormatString :=	'Derotator Axis Error: %s',
	OnMessage := 	NCError_TO_STRING(ErrorID),
	OffMEssage := 	'OK',
	OffLevel := 	ADSLOG_MSGTYPE_HINT);
	
TorqueWarning(	
	Trigger := 		TorqueError.Q, 
	Level := 		ADSLOG_MSGTYPE_WARN,
	FormatString :=	'%s',
	OnMessage := 	'Derotator torque is high.');

CalibrationEvent(	
	Trigger := 		Calibrated, 
	Level := 		ADSLOG_MSGTYPE_HINT,
	OnMessage := 	'Derotator is calibrated.');

END_PROGRAM

// ---- POUs/Functions/F_DerotatorPosition2.TcPOU
FUNCTION F_DerotatorPosition2 : LREAL
VAR_INPUT
	// azimuth of the target
	azimuth: LREAL;
	// elevation of the target in degrees
	elevation: LREAL;
	// declination of the target in degrees
	declination: LREAL;
	// latitude in degrees
	latitude:	LREAL;
END_VAR
VAR
	// parallactic angle
	sinpa, de, az, el, la: LREAL;
	parallactic_angle:	LREAL;
	zenith_distance: LREAL;
END_VAR
VAR CONSTANT
	d2r:	LREAL := PI/180.0;
	r2d:	LREAL := 180.0/PI;
	//h2r:	LREAL := PI/12.0;
	//h2d:	LREAL := 15.0;
END_VAR

// calculate the parallactic angle
de := LIMIT(-90.0, declination, 90.0) * d2r;
az := MODABS(azimuth, 360.0) * d2r;
el := LIMIT(0.0, elevation, 90.0) * d2r;
la := LIMIT(-90.0, latitude, 90.0) * d2r;
IF ABS(COS(de)) > 1E-3 THEN
	sinpa := SIN(az) * COS(la) / COS(de);
	parallactic_angle := r2d * ASIN(LIMIT(-1.0, sinpa, 1.0));
ELSE
	// WARNING: arbitrary definition
	parallactic_angle := 0.0;
END_IF
zenith_distance := 90.0 - elevation;
F_DerotatorPosition2 := parallactic_angle + azimuth - zenith_distance;

END_FUNCTION

// ---- POUs/Functions/F_Derotatorvelocity.TcPOU
FUNCTION F_Derotatorvelocity : LREAL
VAR_INPUT
	// elevation in degrees
	elevation: 	LREAL;
	// azimuth in degrees
	azimuth:	LREAL;
	// observers latitude in degrees
	latitude:	LREAL;
END_VAR
VAR
END_VAR
VAR CONSTANT
	// Earth's angular rotation frequency in [deg/s]
	Omega: LREAL := 4.178E-3;
	d2r:	LREAL := PI/180.0;
	//r2d:	LREAL := 180.0/PI;
END_VAR

(* 
source: https://github.com/cytan299/field_derotator/blob/master/field_derotator_formula/field_derotator_formula.pdf
https://circuitcellar.com/research-design-hub/projects/field-derotator-for-astrophotography-part-1/

returns the rotational velocity for the de-rotator in degrees per second
azimuth, latitutde and elevation are converted to radians
*)
IF ABS(COS(elevation * d2r))> 1.0e-3 THEN
	F_Derotatorvelocity := -Omega * COS(azimuth * d2r) * COS(latitude * d2r) / COS(elevation * d2r);
ELSE
	F_Derotatorvelocity := 0.0;	
END_IF

END_FUNCTION

// ---- POUs/PendantControl.TcPOU
PROGRAM PendantControl
VAR
	// program selection of the pendant control
	Selection:	UINT;
	// error on the pendant control
	Error:		BOOL;
	// manual switch
	manual:		BOOL;
	//enable button
	enable:		BOOL;
	//reset button
	reset:		BOOL;
	// up button
	up:			BOOL;
	// down button
	down:		BOOL;
	// left button
	left:		BOOL;
	// right button
	right:		BOOL;
	lamp_left:		BOOL;
	lamp_right:		BOOL;
	lamp_up:		BOOL;
	lamp_down:		BOOL;
	lamp_error:		BOOL;
	horn:			BOOL;
	// counter for filter position
	Filter_position:	CTUD;
	CoverEnable: FB_ButtonEnable;
	NasmythEnable: FB_ButtonEnable;
	FocusEnable: FB_ButtonEnable;
	DerotatorEnable:	FB_ButtonEnable;
	ElevationEnable: 	FB_ButtonEnable;
	AzimuthEnable: 		FB_ButtonEnable;
	TelescopeControlEnable: 	FB_ButtonEnable;
	HydraulicsEnable: 	FB_ButtonEnable;
	TrackingEnable:			FB_ButtonEnable;
	ResetDelay:	TON;
	TwinCATRestart: TC_Restart;
	//R_Enable:	R_TRIG;
END_VAR

(* 
This program is responsible for the manual control of the telescope.
all movable parts can be controlled from here. This is mainly for testing and
maintenance.
WARNING! Some of the safety routines are disabled, when operating the telescope manually.
*)
// calculate the value of the selector
Selection := 1*BOOL_TO_UINT(GVL_pendant_control.BCD1) + 
			 2*BOOL_TO_UINT(GVL_pendant_control.BCD2) + 
			 4*BOOL_TO_UINT(GVL_pendant_control.BCD4) +
			 8*BOOL_TO_UINT(GVL_pendant_control.BCD8);

// detect disconnection of the manual controls (should also trigger emergency stop).			 
Error := (Selection = 0);

// disable all the lamps
lamp_left := FALSE;
lamp_right := FALSE;
lamp_up := FALSE;
lamp_down := FALSE;
horn := FALSE;

// clooect the state of all buttons
manual := GVL_pendant_control.key_switch;
enable := GVL_pendant_control.start_switch;
reset := GVL_pendant_control.reset_switch;
up := GVL_pendant_control.direction_up;
down := GVL_pendant_control.direction_down;
left := GVL_pendant_control.direction_left;
right := GVL_pendant_control.direction_right;

//R_Enable(CLK := enable);
// the error lamp is the same as the error lamp of the main panel
lamp_error := GVL_Main.lamp_error;
CoverControl.active_cover := 0;
// enable only the selected item and connect lamps and buttons accordingly
CASE Selection OF
	1:	// reserved for Cover1 control

	2: // Cover2 control
		lamp_up := GVL_Telescope.cover2_open AND CoverControl.Ready;
		lamp_down := GVL_Telescope.cover2_closed AND CoverControl.Ready;
		IF manual THEN
			CoverEnable(SET := enable, Q := CoverControl.enable);
			CoverControl.active_cover := 2;
			CoverControl.reset := reset;
			CoverControl.open := up AND CoverControl.Ready;
			CoverControl.close := down AND CoverControl.Ready;
			lamp_error := CoverControl.Cover2_Error;
		END_IF
 	
	3:  // Cover3 control
		lamp_up := GVL_Telescope.cover3_open AND CoverControl.Ready;
		lamp_down := GVL_Telescope.cover3_closed AND CoverControl.Ready;
		IF manual THEN
			CoverEnable(SET := enable, Q := CoverControl.enable);
			CoverControl.active_cover := 3;
			CoverControl.open := up AND CoverControl.Ready;
			CoverControl.close := down AND CoverControl.Ready;
			CoverControl.reset := reset;
			lamp_error := CoverControl.Cover3_Error;
		END_IF
		
	4:	// Nasmyth / mirror M3 control
		lamp_left := GVL_Telescope.nasmyth_limit_left AND NasmythControl.Ready;
		lamp_right := GVL_Telescope.nasmyth_limit_right AND NasmythControl.Ready;
		IF manual THEN
			NasmythEnable(SET := enable, Q := NasmythControl.enable);
			NasmythControl.left := left;
			NasmythControl.right := right;
			NasmythControl.reset := reset;
			lamp_error := Nasmythcontrol.error;
		END_IF
		
	5:	// Focus Control
		lamp_up := FocusControl.Ready AND NOT GVL_Telescope.focus_limit_far;
		lamp_down := FocusControl.Ready AND NOT GVL_Telescope.focus_limit_near;
		IF manual THEN
			FocusEnable(SET := enable, Q := FocusControl.enable);
			FocusControl.outward := up;
			FocusControl.inward := down;
			Focuscontrol.reset := reset;
			lamp_error := FocusControl.error;
		END_IF
							
	6:	// Derotator control
		lamp_left := DerotatorControl.Ready AND NOT GVL_Telescope.Derotator_inputs.1;
		lamp_right :=DerotatorControl.Ready AND NOT GVL_Telescope.Derotator_inputs.0;
		IF manual THEN
			DerotatorEnable(SET := enable, Q := DerotatorControl.enable);
			DerotatorControl.left := left AND NOT GVL_Telescope.Derotator_inputs.1;
			DerotatorControl.right := right AND NOT GVL_Telescope.Derotator_inputs.0;
			DerotatorControl.reset := reset;
			lamp_error := DerotatorControl.Error;
		END_IF
							
	7:	// Elevation Control
		
		ElevationControl.up := up AND GVL_Telescope.Elevation_inputs.0;
		ElevationControl.down := down AND GVL_Telescope.Elevation_inputs.1;
		IF manual THEN
			ElevationEnable(
				SET := enable, 
				Q := ElevationControl.enable);	
		END_IF
		ElevationControl.reset := reset;
		lamp_up := GVL_Telescope.Elevation_inputs.0;
		lamp_down := GVL_Telescope.Elevation_inputs.1;
		lamp_error := ElevationControl.error;
		
	8:	// Azimuth Control
		lamp_left := GVL_Telescope.Azimuth_inputs.0; // NOT GVL_Telescope.azimut_limit_switch;
		lamp_right := GVL_Telescope.Azimuth_inputs.1; // NOT GVL_Telescope.azimut_limit_switch;
		AzimuthElevationControl.left := left AND GVL_Telescope.Azimuth_inputs.0;
		AzimuthElevationControl.right := right AND GVL_Telescope.Azimuth_inputs.1;
		AzimuthElevationControl.reset := reset;
		IF manual THEN
			AzimuthEnable(
				SET := enable, 
				Q := AzimuthElevationControl.enable);
			lamp_error := AzimuthElevationControl.error;
		END_IF
		
	9: 	// Dome control
		DomeControl.left := left;
		DomeControl.right := right;
		DomeControl.OpenDome := up;
		DomeControl.CloseDome := down;
		DomeControl.reset := reset;
		lamp_left := DomeControl.enable;
		lamp_right := DomeControl.enable;
		lamp_up := DomeControl.DomeClosed;
		lamp_down := DomeControl.DomeOpened;
		IF manual THEN
			lamp_error := DomeControl.Error;
		END_IF
		
		
	10:	// FilterWheel control
		//FIXME
		FilterWheelControl.Enable := manual;
		lamp_left := manual;
		lamp_right := manual;
		FilterWheelControl.left := left;
		FilterWheelControl.right := right;
		Filter_position(CU := up, CD := down, RESET := reset, PV := 15);
		lamp_up := NOT Filter_position.QU;
		lamp_down := NOT Filter_position.QD;
		IF enable THEN
			FilterWheelControl.filter_position := Filter_position.CV;
		END_IF
		FilterWheelControl.reset := reset;
		IF manual THEN
			lamp_error := FilterWheelControl.Error;
		END_IF
		
	11: horn := manual;
		
	12:	// manual Telescope Control
		IF manual THEN
			lamp_up := TelescopeControl.power;
			lamp_down := TelescopeControl.power;
			lamp_left := TelescopeControl.power;
			lamp_right := TelescopeControl.power;
	
			TelescopeControl.gohome := down;
			TelescopeControl.park := up;
			TelescopeControl.goto := right;
			TrackingEnable(SET := enable, 
							RESET := reset, 
							Q := TelescopeControl.track);
			TelescopeControl.reset := reset;
			Telescopecontrol.stop := left;	
			lamp_error := Telescopecontrol.error;
		END_IF
		
	13: // Telescope Control
		TelescopeControlEnable(
			SET := enable, 
			Q := TelescopeControl.power);
		TelescopeControl.reset := reset;
		IF manual THEN
			lamp_up := GVL_Telescope.Elevation_inputs.0;
			lamp_down := GVL_Telescope.Elevation_inputs.1;
			lamp_left := GVL_Telescope.Azimuth_inputs.0;
			lamp_right := GVL_Telescope.Azimuth_inputs.1;
			ElevationControl.up := up AND GVL_Telescope.Elevation_inputs.0;
			ElevationControl.down := down AND GVL_Telescope.Elevation_inputs.1;
			AzimuthElevationControl.left := left AND GVL_Telescope.Azimuth_inputs.0;
			AzimuthElevationControl.right := right AND GVL_Telescope.Azimuth_inputs.1;
			TelescopeControl.rightascension := TelescopeControl.rightascension_calc;
			TelescopeControl.declination := TelescopeControl.declination_calc;
		ELSE
			lamp_up := ElevationControl.enable;
			lamp_down := ElevationControl.enable;
			lamp_left := AzimuthElevationControl.enable;
			lamp_right := AzimuthElevationControl.enable;
			IF up THEN 
				Telescopecontrol.elevation_offset := Telescopecontrol.elevation_offset + 10.0/3600.0; 
			ELSIF down THEN 
				Telescopecontrol.elevation_offset := Telescopecontrol.elevation_offset - 10.0/3600.0; 
			END_IF;
			IF left THEN 
				Telescopecontrol.azimuth_offset := Telescopecontrol.azimuth_offset - 10.0/3600.0; 
			ELSIF right THEN 
				Telescopecontrol.azimuth_offset := Telescopecontrol.azimuth_offset + 10.0/3600.0; 
			END_IF;
		END_IF
		ResetDelay(IN := reset, PT := T#3S);
		// wait for suction pump to stop
		TwinCATRestart(NETID := '', RESTART := ResetDelay.Q AND NOT HydraulicsControl.suction_running, TMOUT := T#60S);
	
	14: horn := manual;
	
	15:	// Hydraulics control
		lamp_up := HydraulicsControl.oil_pressure_OK AND Hydraulicscontrol.brake_closed;
		lamp_down := HydraulicsControl.oil_pressure_OK AND Hydraulicscontrol.brake_open;
		lamp_left := HydraulicsControl.pump_running;
		lamp_right := HydraulicsControl.suction_running;
		IF manual THEN
			HydraulicsEnable(
				SET := enable, 
				Q := Hydraulicscontrol.start);
			Hydraulicscontrol.stop := NOT Hydraulicscontrol.start;
			Hydraulicscontrol.reset := reset;
			
			IF up THEN
				Hydraulicscontrol.open_brake := TRUE;
				Hydraulicscontrol.close_brake := FALSE;
			END_IF
			IF down THEN
				Hydraulicscontrol.open_brake := FALSE;
				Hydraulicscontrol.close_brake := TRUE;
			END_IF
			lamp_error := HydraulicsControl.error;
		END_IF
END_CASE

// set all the lamps
GVL_pendant_control.lamp_left := lamp_left;
GVL_pendant_control.lamp_right := lamp_right;
GVL_pendant_control.lamp_up := lamp_up;
GVL_pendant_control.lamp_down := lamp_down;
GVL_pendant_control.lamp_error := lamp_error;

END_PROGRAM

// ---- POUs/CoverControl.TcPOU
PROGRAM CoverControl
VAR_INPUT
	// enables all cover drivers
	enable:		BOOL;
	// resets all drives after an error has occured
	reset:		BOOL;
	// open the cover in proper order
	open:		BOOL;
	// close the cover in proper order
	close:		BOOL;
	// actual active cover in manual mode, 0 for automatic = all covers active
	active_cover:	INT;

END_VAR
VAR_OUTPUT
	// is TRUE, if all covers are open
	isopen:			BOOL;
	// is TRUE, if all covers are closed
	isclosed:		BOOL;
	// is TRUE if any cover-driver reports an error
	Error: 	BOOL;
	// warning state of the DC drives
	Warning: BOOL;
	// cover2 is open
	Cover2_opened, 
	// cover2 is closed
	Cover2_closed:	BOOL;
	// cover3 is open
	Cover3_opened, 
	// cover3 is closed
	Cover3_closed:	BOOL;
	Cover2_error: BOOL;
	Cover3_error: BOOL;
	Ready:		BOOL;
END_VAR
VAR
	// delay timer for opening cover2
	open2_delay: 	TON;
	// dely timer for closing cover3
	close3_delay : 	TON;
	
	//Cover3_state: 	RS;
	//triggers for timeout event for cover1
	Cover2_timeout,
	Cover3_timeout:	TON;
	error_trigger: SR;
	//error event for cover
	Cover2_Event,
	Cover3_Event:	FB_EventLog;
	// timeout event for cover1
	Cover2_Timeout_Event,
	Cover3_Timeout_Event:	FB_EventLog;
	// log if covers are open
	Covers_opened_event,
	// log if covers are closed
	Covers_closed_event:	FB_EventLog;
	// Event log for a generic drive error
	Covers_Error_event:		FB_EventLog;
	// Event log for a generic drive warning
	Covers_Warning_event:		FB_EventLog;
	// status word for MQTT message
	Cover_status:		WORD;
	// last status word to trigger MQTT message if different
	LastStatus:			WORD;
END_VAR

(*
This is the control for the two (three) telescope covers. 
The correct order for opening is 1->3->2 and for closing 2->3->1.
GVL Open and close signals are inverted
*)

// close has precedence over open
IF close THEN
	open := FALSE;
END_IF

IF Error THEN
	open := FALSE;
	close := FALSE;
END_IF

Cover2_opened := NOT GVL_Telescope.cover2_open;
Cover3_opened := NOT GVL_Telescope.cover3_open;
Cover2_closed := NOT GVL_Telescope.cover2_closed;
Cover3_closed := NOT GVL_Telescope.cover3_closed;

IF active_cover = 2 THEN
	GVL_Telescope.open_cover2 := enable AND open AND NOT Cover2_opened;
	GVL_Telescope.close_cover2 := enable AND close AND NOT Cover2_closed;
ELSIF active_cover = 3 THEN
	GVL_Telescope.open_cover3 := enable AND open AND NOT Cover3_opened;
	GVL_Telescope.close_cover3 := enable AND close AND NOT Cover3_closed;
ELSE
	// we open both covers
	// wait for cover2 until cover3 has left the closed state
	open2_delay(IN := enable AND open AND NOT cover3_closed,
				PT := T#300MS);
	// wait for cover3 until cover2 has left the open state
	close3_delay(IN := enable AND close AND NOT cover2_opened,
				PT := T#1500MS);
	GVL_Telescope.open_cover2 := enable AND open AND open2_delay.Q AND NOT Cover2_opened;
	GVL_Telescope.open_cover3 := enable AND open AND NOT Cover3_opened;
	
	GVL_Telescope.close_cover2 := enable AND close AND NOT Cover2_closed;
	GVL_Telescope.close_cover3 := enable AND close AND close3_delay.Q AND NOT Cover3_closed;
END_IF

